# B&R Automation Studio project CombinedLinenSoiledA9KAN (part 17)

#### KanLinkCyclic.st - Cyclic code
```iecst
(********************************************************************
 * COPYRIGHT -- Herbert Kannegiesser GmbH
 ********************************************************************
 * Program: KanLink
 * File: KanLinkCyclic.st
 * Author: stahlhut
 * Created: December 23, 2011
 ********************************************************************
 * Implementation of program WetLink
 ********************************************************************)

(*
	todo
			logger !

	Mögliche Fehler
	1= Configuration kann nicht gelesen werden
	2= Port kann nicht geöffnet werden
	4= Fehler bei UDPSend
	5= Fehler bei UDPRec
*)

PROGRAM _CYCLIC

	// ===========================
	// Logging
	// ===========================

	IF _xRBReady THEN

		CASE _wLogStep OF

			0:
				_ReadRB(wPtrRead := _wPtrRBread, wPtrStart := _wPtrRBstart, wPtrWrite := _wPtrRBwrite);

				IF _ReadRB.wStatus = ERR_OK THEN

					CASE _LogEntry.wErrorNo OF

						0:
							_kgArLogWrite.text := 'OK';

						HLKANLINK_MSG_NO_STRUCDEF:

							_kgArLogWrite.text := 'Create Strucdefinition failed : {##AttrVar1} / {##AttrVar2}';
							_kgArLogWrite.var1 := _LogEntry.lAttr1;

						ELSE

							_kgArLogWrite.text := UINT_TO_STRING(_LogEntry.wErrorNo);
							_kgArLogWrite.text := CONCAT(_kgArLogWrite.text, ' : {##AttrVar1} / {##AttrVar2}');
							_kgArLogWrite.var1 := _LogEntry.lAttr1;
							_kgArLogWrite.var2 := _LogEntry.lAttr2;

					END_CASE

					_wLogStep := 1;

				END_IF

			1:
				_kgArLogWrite();

				IF _kgArLogWrite.status <> ERR_FUB_BUSY THEN

					_wLogStep := 0;

				END_IF

		END_CASE

	END_IF

	IF _wDebIdx >= 0 AND _wDebIdx <= _HLKANLINK_MAX_IDX_DEFSTRUC THEN

		IF _lPtrStrucDef[_wDebIdx] > 0 THEN

			_sDebString ACCESS _lPtrStrucDef[_wDebIdx] + _wDebOffset;

		END_IF

	END_IF

	// =======================================================================
	// =======================================================================

	IF _xInitOK THEN

		IF _xSaveConfig THEN
			KL_SaveConfDO_0(adrName :=ADR('KL_Conf') , adrDaten := ADR(IFhlKanLink.Parameter), len := SIZEOF( IFhlKanLink.Parameter));
			IF KL_SaveConfDO_0.status <> ERR_FUB_BUSY THEN // fertig
				_xSaveConfig := FALSE;
			END_IF;
		END_IF;

		IF EDGEPOS(IFhlKanLink.in.xRun ) THEN
			IF Kanlink.Step = 0 THEN
				Kanlink.Step := 1;
			END_IF;
		END_IF;
		IF EDGENEG(IFhlKanLink.in.xRun) THEN // stoppen
			IF Kanlink.Step <> 0 THEN
				Kanlink.Step := 20;
			END_IF;
		END_IF;

		IF IFhlKanLink.in.xRestart THEN
			Kanlink.Step := 1;
			IFhlKanLink.in.xRestart := 0;
		END_IF;

		IFhlKanLink.xError := (Kanlink.Step = 200);

		CASE Kanlink.Step OF

			0: //nix tun

			100: // Error nr in Logger eintragen

				Kanlink.Step := 200;

			200: // Auf User warten

			1: // init

				Kanlink.KLLib_Init_0(enable := 1, adrServer := ADR(Kanlink),adrInterface := ADR(IFhlKanLink));
				IF Kanlink.KLLib_Init_0.status = ERR_OK THEN
					Kanlink.Step := 10;
				ELSIF Kanlink.KLLib_Init_0.status <> ERR_FUB_BUSY THEN // fehler
					WL_ErrorNr := 10;
					Kanlink.Step := 100;

					IF _xRBReady THEN

						_LogEntryIn.wErrorNo := 10;
						_InsertRB(wPtrStart := _wPtrRBstart, wPtrRead := _wPtrRBread, wPtrWrite := _wPtrRBwrite);

					END_IF

				END_IF;

			10: // Kanlink Run

			20: // Kanlink schliessen
				Kanlink.UdpClose_0(enable := 1);
				Kanlink.UdpClose_0.enable := 1;
				Kanlink.UdpClose_0.ident := Kanlink._uiLastId;
				Kanlink.UdpClose_0;
				IF Kanlink.UdpClose_0.status = 0 THEN
					Kanlink.Step := 0;
				ELSIF Kanlink.UdpClose_0.status = ERR_FUB_BUSY THEN

				ELSE
					Kanlink.Step := 100;
				END_IF;

		END_CASE;

		// hier beenden wenn zyklus nicht erlaubt
		IF  Kanlink.Step <> 10 THEN
			RETURN;
		END_IF;

		//
		// Client Timeout bearbeiten

		Kanlink;

		IF Kanlink.xReturn THEN
			RETURN;
		END_IF;

		IF Kanlink._xGetServerReq THEN  // ServerReq angenommen, bearbeiten

			// antwort zusammenbauen

			// Commandos unter 1000 sind für alle gleich:
			IF Kanlink.ServerData.HeaderV1Rec.Command < 1000 THEN

				CASE Kanlink.ServerData.HeaderV1Rec.Command OF
					0:   // MaschinenInfo Senden: Darf jeder lesen

						Kanlink.ServerData.HeaderV1Send.Command := 1;
						Kanlink.ServerData.HeaderV1Send.dataFormat := 5;
						Kanlink.ServerData.HeaderV1Send.Length := 148;
						Kanlink.ServerData.HeaderV1Send.Tag := Kanlink.ServerData.HeaderV1Rec.Tag;
						Kanlink.ServerData.HeaderV1Send.ReqID := Kanlink.ServerData.HeaderV1Rec.ReqID;

						KLLib_SendData(ADR(Kanlink),ADR(Kanlink.ServerData.MetaInfoResp),SIZEOF(Kanlink.ServerData.MetaInfoResp),ADR(Kanlink.client_address));

					2:   // Response Ping: Darf jeder lesen

						Kanlink.ServerData.HeaderV1Send.Command := 3;
						Kanlink.ServerData.HeaderV1Send.dataFormat := 5;
						Kanlink.ServerData.HeaderV1Send.Length := 17;
						Kanlink.ServerData.HeaderV1Send.Tag := Kanlink.ServerData.HeaderV1Rec.Tag;
						Kanlink.ServerData.HeaderV1Send.ReqID := Kanlink.ServerData.HeaderV1Rec.ReqID;

						KLLib_SendData(ADR(Kanlink),ADR(Kanlink.ServerData.PingResp),SIZEOF(Kanlink.ServerData.PingResp),ADR(Kanlink.client_address));

				END_CASE;

			ELSE
					// >= 1000 sind spezifische Daten

					// Anfrage Konfiguriert?
					// Zur Anfrage Verbindung raussuchen..
					_xIdxFound := FALSE;
					_iIdxFound := 32000;

					//Kanlink.udRecKey	:= SHL(UINT_TO_UDINT( Kanlink.ServerData.HeaderV1Rec.Command),16)  + SHL(USINT_TO_UINT( Kanlink.ServerData.recArea),8) + Kanlink.ServerData.recAddr;

					Kanlink.udRecKey := KL_BuildKey(Command := Kanlink.ServerData.HeaderV1Rec.Command,CmdNr := UINT_TO_USINT( Kanlink.ServerData.HeaderV1Rec.CmdNr AND 16#000F) ,Area := Kanlink.ServerData.recArea,IPAdr:= Kanlink.ServerData.recAddr);
					FOR _i := 0 TO HLKANLINK_MAX_SERVERCONNS  DO

						_ptrIndex ACCESS ADR(Kanlink.ServerListe[_i]);
						_dSrvIf ACCESS _ptrIndex.adrInterface;
						_udRecKey := Kanlink.udRecKey;
						IF _ptrIndex.Adr = 0 THEN // wenn alle das Commando lesen dürfen/ Adresse und Area ausblenden
							_udRecKey := Kanlink.udRecKey AND 16#FFFF_0000;
						END_IF;
						IF _udRecKey = _ptrIndex.Key THEN // Index gefunden, beantworten:
							_xIdxFound := TRUE;
							_iIdxFound := _i;
							EXIT;
						END_IF;
					END_FOR

					_xAdrErr := (_ptrIndex.AdrDataReq = 0) OR (_ptrIndex.AdrDataResp = 0);

					IF ( _xIdxFound = FALSE) OR _xAdrErr THEN // Falls keine gültige Verbindung dann Fehlerframe senden
						// Fehlerframe senden:
						Kanlink.ServerData.HeaderV1Send.Command := Kanlink.ServerData.HeaderV1Rec.Command +1;
						Kanlink.ServerData.HeaderV1Send.dataFormat := 255;
						Kanlink.ServerData.HeaderV1Send.Length := 68;
						Kanlink.ServerData.HeaderV1Send.Tag := Kanlink.ServerData.HeaderV1Rec.Tag;
						Kanlink.ServerData.HeaderV1Send.ReqID := Kanlink.ServerData.HeaderV1Rec.ReqID;

						// Error Frame:
						Kanlink.ServerData.ErrorFrame.ErrorNumber := 2;
						strcpy(ADR(Kanlink.ServerData.ErrorFrame.ErrorText),ADR('request not supported'));

					//	KLLib_SendData(ADR(Kanlink),ADR(Kanlink.ServerData.ErrorFrame),SIZEOF(Kanlink.ServerData.ErrorFrame),ADR(Kanlink.client_address));

				ELSE
						// Empfangene Daten speichern:

						IF NOT( (_dSrvIf.iState <> 0 )   AND _ptrIndex.xReqManually) THEN  // falls Req bereits bearbeitet wird verwerfen
							_ptrIndex.iReqCnt := _ptrIndex.iReqCnt + 1;
							_dSrvIf.iState := 1;
							strcpy(ADR(_ptrIndex.sClientIPAdr),ADR(Kanlink.client_address));
							// todo längenüberprüfung _ptrIndex.ReqLength
							memcpy(_ptrIndex.AdrDataReq,ADR(Kanlink.ServerData.receive_data)+PreHeaderSize+HeaderSize,_ptrIndex.ReqLength);

							_ptrIndex.iReqID := Kanlink.ServerData.HeaderV1Rec.ReqID;
							IF (_ptrIndex.CmdOpt AND KL_optOnReqCall) <> 0 THEN
								KL_OnRecReq(adrReqData := _ptrIndex.AdrDataReq, adrRespData := _ptrIndex.AdrDataResp, adrKanlink := ADR(Kanlink),_ptrIndex.Cmd, adrUserData := IFhlKanLink.Parameter.adrUserTyp );
							END_IF;
							IF _ptrIndex.xReqManually = 0 THEN

								Kanlink.ServerData.HeaderV1Send.Command := _ptrIndex.Cmd + 1;
								Kanlink.ServerData.HeaderV1Send.dataFormat := 5;
								Kanlink.ServerData.HeaderV1Send.Length := UDINT_TO_UINT( _ptrIndex.RespLength);
								Kanlink.ServerData.HeaderV1Send.ReqID := _ptrIndex.iReqID;
								Kanlink.ServerData.HeaderV1Send.CmdNr := _ptrIndex.CmdOpt AND 16#000F;
								_ptrIndex.iConnectionTimer := 0;
								KLLib_SendData(ADR(Kanlink),_ptrIndex.AdrDataResp,_ptrIndex.RespLength,ADR(_ptrIndex.sClientIPAdr));
							END_IF;
						END_IF;

					END_IF;

			END_IF;

			Kanlink._xGetServerReq := FALSE;
			Kanlink.UdpRecv_0.enable := 1;

			RETURN;  // Daten sind versendet. Also Ende.

		END_IF;

		IF Kanlink._xGetClientResp THEN // Response auf ClientReq angekommen

			Kanlink.udRecKey := KL_BuildKey(Command := Kanlink.ServerData.HeaderV1Rec.Command,CmdNr := UINT_TO_USINT( Kanlink.ServerData.HeaderV1Rec.CmdNr AND 16#000F) ,Area := Kanlink.ServerData.recArea,Kanlink.ServerData.recAddr);

			_xIdxFound := FALSE;
			FOR _i := 0 TO HLKANLINK_MAX_CLIENTCONNS DO
				_dClient ACCESS ADR(Kanlink.ClientListe[_i]);
					//Kanlink.udRecKey 	:= SHL(UINT_TO_UDINT( Kanlink.ServerData.HeaderV1Rec.Command),16)  + SHL(USINT_TO_UINT( Kanlink.ServerData.recArea),8) + Kanlink.ServerData.recAddr;

					IF Kanlink.udRecKey = _dClient.Key THEN // Index gefunden, beantworten:
						_xIdxFound := TRUE;
					EXIT;
				END_IF;
			END_FOR

			_xAdrOK := _dClient.AdrDataResp <> 0 ;

			IF _xIdxFound AND _xAdrOK THEN
				_dClient.xReqPending := FALSE;
				IF _dClient.iTimeOutCnt > 0 THEN
					_dClient.iTimeOutCnt := _dClient.iTimeOutCnt - 1;
				END_IF;
				IF _dClient.adrInterface <> 0 THEN
					_dCltIf ACCESS _dClient.adrInterface;
					_dCltIf.iState := 3;
				END_IF;

				memcpy(_dClient.AdrDataResp,ADR(Kanlink.ServerData.receive_data) + PreHeaderSize+HeaderSize,_dClient.RespLength);

		  	END_IF;

			_iCltRespCnt := _iCltRespCnt + 1;
			Kanlink._xGetClientResp := FALSE;

			Kanlink._xSendClient := TRUE; // Daten einsortiert, nix weiter zutun also Clients bearbeiten
			Kanlink.UdpRecv_0.enable := 1;

		END_IF;

		// Überprüfen ob per Hand bearbeitete Requests versendet werden müssen..

		IF  Kanlink.UdpSend_0.enable = 0 THEN
			_xServerFound := 0;

			FOR _i:=0 TO HLKANLINK_MAX_SERVERCONNS  DO
				_ptrIndex ACCESS ADR(Kanlink.ServerListe[_iLastServerIdx]);
				_dSrvIf ACCESS _ptrIndex.adrInterface;
				IF (_ptrIndex.xReqManually AND (_dSrvIf.iState = 2)) THEN
					_xServerFound := 1;

					_iLastServerIdx := _iLastServerIdx + 1; // testen
					IF _iLastCltIdx > HLKANLINK_MAX_SERVERCONNS THEN
						_iLastServerIdx := 0;
					END_IF;
					EXIT;
					END_IF;
					_iLastServerIdx := _iLastServerIdx + 1; // testen
					IF _iLastServerIdx > HLKANLINK_MAX_SERVERCONNS THEN
					_iLastServerIdx := 0;
				END_IF;

			END_FOR;

			IF _xServerFound THEN

				Kanlink.ServerData.HeaderV1Send.Command := _ptrIndex.Cmd + 1;
				Kanlink.ServerData.HeaderV1Send.dataFormat := 5;
				Kanlink.ServerData.HeaderV1Send.Length := UDINT_TO_UINT( _ptrIndex.RespLength);
				Kanlink.ServerData.HeaderV1Send.ReqID := _ptrIndex.iReqID;
				Kanlink.ServerData.HeaderV1Send.CmdNr := _ptrIndex.CmdOpt AND 16#000F;
				_ptrIndex.iConnectionTimer := 0;
				KLLib_SendData(ADR(Kanlink),_ptrIndex.AdrDataResp,_ptrIndex.RespLength,ADR(_ptrIndex.sClientIPAdr));
				_dSrvIf.iState := 0;
				RETURN;
			END_IF;
		END_IF;

		IF Kanlink._xSendClient THEN  // hier den Clienten bearbeiten

			_xCltFound := FALSE;

			FOR _i:=0 TO HLKANLINK_MAX_CLIENTCONNS  DO
				_dClient ACCESS ADR(Kanlink.ClientListe[_iLastCltIdx]);
				IF _dClient.adrInterface <> 0 THEN
					_dCltIf ACCESS _dClient.adrInterface;
				ELSE
					_dCltIf ACCESS ADR(_ifDummy);
				END_IF;
					// gefunden wenn kein ReqPend, Commando <> 0 todo gültige Adresse etc...
				IF _dClient.iCycleTime = 0 THEN
					_xSendNow := (_dCltIf.iState = 1) OR (_dCltIf.iState = 4) ; // falls angetickt oder timeout
				ELSE
					_xSendNow := (_dClient.iCycleWait > _dClient.iCycleTime);
				END_IF;
				IF 	(NOT _dClient.xReqPending) AND (_dClient.Cmd <> 0) AND  _dClient.xActiv AND (_xSendNow)   THEN
		  			_xCltFound := TRUE;
					_iLastCltIdx := _iLastCltIdx + 1; // testen
					IF _iLastCltIdx > HLKANLINK_MAX_CLIENTCONNS THEN
			  			_iLastCltIdx := 0;
					END_IF;
					EXIT;
				END_IF;

				_iLastCltIdx := _iLastCltIdx + 1; // testen
				IF _iLastCltIdx > HLKANLINK_MAX_CLIENTCONNS THEN
		  			_iLastCltIdx := 0;
				END_IF;

			END_FOR;

			IF NOT _xCltFound THEN
				Kanlink._xSendClient := FALSE;
				RETURN;

			ELSE

				// Client gefunden
				_dClient.iCnt := _dClient.iCnt + 1 ;
				_dClient.iReqId := _dClient.iReqId +1;
				_dClient.TimeOutLeft := _dClient.TimeOut;

				IF _dCltIf.iState = 1 THEN // falls über state dann "schnellwiederholung" aktivieren
					_dClient.iTimeOutCnt := 0; // scharf machen für den nächsten versuch
				END_IF;
				_dCltIf.iState := 2;

				Kanlink.ServerData.HeaderV1Send.Command := _dClient.Cmd;
				Kanlink.ServerData.HeaderV1Send.CmdNr := _dClient.CmdOpt AND 16#000F;

				Kanlink.ServerData.HeaderV1Send.dataFormat := 5;
				Kanlink.ServerData.HeaderV1Send.Length := UDINT_TO_UINT( _dClient.ReqLength);
				Kanlink.ServerData.HeaderV1Send.ReqID := _dClient.iReqId;

				KLLib_SendData(ADR(Kanlink),_dClient.AdrDataReq,_dClient.ReqLength,ADR(_dClient.sClientAdr));

				_dClient.xReqPending := TRUE;
				_dClient.iCycleWait := 0;

				Kanlink._xSendClient := FALSE;

				RETURN;

			END_IF;

		END_IF;	// sendClient

	ELSIF IFmnParam.Out.xParamOK AND IFmnEth.Out.xDataValid THEN

		Kanlink.ServerData.MetaInfoResp.KanLink_Hostname := IFmnEth.Out.IP.sHostname;
		Kanlink.ServerData.MetaInfoResp.Machine_type := WSTRING_TO_STRING(IFmnParam.Out.HeaderVersion.utfMachineType);
		Kanlink.ServerData.MetaInfoResp.DataModelTimeStamp := IFmnParam.Out.HeaderVersion.dtTimestamp;
		Kanlink.ServerData.MetaInfoResp.DataModelVersion := IFmnParam.Out.HeaderVersion.wVersion;

		Kanlink.ServerData.PingResp.KanLink_Hostname := IFmnEth.Out.IP.sHostname;

		_xInitOK := TRUE;

	END_IF

END_PROGRAM
```

#### KanLinkInit.st - Initialization code
```iecst
(********************************************************************
 * COPYRIGHT -- Herbert Kannegiesser GmbH
 ********************************************************************
 * Program: KanLink
 * File: KanLinkInit.st
 * Author: stahlhut
 * Created: December 23, 2011
 ********************************************************************
 * Implementation of program KanLink
 ********************************************************************)

PROGRAM _INIT

	// Packet-Version auslesen mit MO_ver aus SYS_lib und für den Additional Status zur Verfügung stellen

	_sPkgName := 'hlKanLink';

	IF ( MO_ver(ADR(_sPkgName), 0, ADR(_VerStruc)) = 0 ) THEN

		brsmemcpy(ADR(hlKanLinkStatAd.sPkgVersion), ADR(_VerStruc.version), SIZEOF(_VerStruc.version));

	ELSE

		hlKanLinkStatAd.sPkgVersion := '---';

	END_IF

	_xInitOK := FALSE;

	// nötige adressen initialisieren:
	Kanlink.adrSelf := ADR(Kanlink);
	Kanlink.CfgServer.adrKanlink := ADR(Kanlink);
	Kanlink.CfgClient.adrKanlink := ADR(Kanlink);

	FOR _i := 0 TO HLKANLINK_MAX_SERVERCONNS DO
		Kanlink.ServerListe[_i].adrInterface := ADR(IFhlKanLink.Server[_i]);
		KLLib_ReadServerPara(ADR(Kanlink.ServerListe[_i]), ADR( IFhlKanLink.Parameter.Server[_i]));
	END_FOR;

	FOR _i := 0 TO HLKANLINK_MAX_CLIENTCONNS DO
		KLLib_ReadClientPara(ADR(Kanlink.ClientListe[_i]),ADR(IFhlKanLink.Parameter.Client[_i]),ADR(Kanlink));
		Kanlink.ClientListe[_i].TimeOut := 140;
		Kanlink.ClientListe[_i].adrInterface := ADR(IFhlKanLink.Parameter.Client[_i]);
	END_FOR;

	// Create Log
	//****************************************************************************************************************
	// Log erzeugen
	//****************************************************************************************************************

	_kgArLogWrite.enable := TRUE;
	_kgArLogWrite.ident := 0;
	_kgArLogWrite.errornr := 50010;

	_AsArLogCreate(enable := TRUE, pName := ADR('hlKanLinkL'), len := 4096*1, memType := arlogUSRROM);

	IF _AsArLogCreate.status = ERR_OK THEN

		_kgArLogWrite.ident := _AsArLogCreate.ident;

	ELSIF _AsArLogCreate.status = arlogERR_EXISTING THEN

		_AsArLogGetInfo(enable := TRUE, pName := ADR('hlKanLinkL'));

		IF _AsArLogGetInfo.status = ERR_OK THEN

			_kgArLogWrite.ident := _AsArLogGetInfo.ident;

		END_IF

	END_IF

	//****************************************************************************************************************
	// Ringbuffer for Logs
	//****************************************************************************************************************

	_kgRBcreateKanLinklog(sName := '_klLogrb', bMemType := doUSRRAM, wCntEntry := 10, lLenEntry := SIZEOF(_LogEntry), wPtrWrite := _wPtrRBwrite, wPtrRead := _wPtrRBread, wPtrStart := _wPtrRBstart);

	IF _kgRBcreateKanLinklog.wStatus = ERR_OK THEN

		_wPtrRBloc := 0;

		_xRBReady := TRUE;

		_InsertRB.doIdent := _kgRBcreateKanLinklog.doIdent;
		_InsertRB.doLen := _kgRBcreateKanLinklog.doLen;
		_InsertRB.lLenEntry := SIZEOF(_LogEntry);
		_InsertRB.pEntry := ADR(_LogEntryIn);

		_ReadRB.doIdent := _kgRBcreateKanLinklog.doIdent;
		_ReadRB.doLen := _kgRBcreateKanLinklog.doLen;
		_ReadRB.lLenEntry := SIZEOF(_LogEntry);
		_ReadRB.pEntry := ADR(_LogEntry);

	ELSE

		_kgArLogWrite.logLevel := arlogLEVEL_INFO;
		_kgArLogWrite.text := 'Create Ringbuffer: {##AttrVar1}';
		_kgArLogWrite.var1 := _kgRBcreateKanLinklog.wStatus;
		_kgArLogWrite.var2 := 0;
		_kgArLogWrite();

	END_IF

	_wLogStep := 0;

	// Create StructureDescriptions
	//****************************************************************************************************************
	// Speicher allokoieren
	//****************************************************************************************************************

	_MemPartCreate(enable := TRUE, len := 8000);

	_LogEntryIn.wErrorNo := HLKANLINK_MSG_NO_STRUCDEF;

	IF _MemPartCreate.status = ERR_OK THEN

		_lTempMemIdent := _MemPartCreate.ident;

		_MemPartCreate(enable := TRUE, len := 8000);

		IF _MemPartCreate.status = ERR_OK THEN

			_lMemIdent := _MemPartCreate.ident;

			_MemAllocTemp(enable := TRUE, ident := _lTempMemIdent, len := 7500);

			IF _MemAllocTemp.status = ERR_OK THEN

				_lAdr := _MemAllocTemp.mem;
				_lLen := _MemAllocTemp.len;

				_wStatus := KLLib_CreateStrucDef(lPtrAdr := ADR(_lAdr), lPtrLen := ADR(_lLen), sRootName := 'hlKanLink:Kanlink.ServerData.MetaInfoResp', sItemName := '', lDataAdr := 0);

				IF _wStatus = ERR_OK THEN

					_MemAlloc(enable := TRUE, ident := _lMemIdent, len := _MemAllocTemp.len - _lLen);

					IF _MemAlloc.status = ERR_OK THEN

						_lPtrStrucDef[_HLKANLINK_IDX_STRUCDEF_RESP_0] := _MemAlloc.mem;
						_lPtrStrucLen[_HLKANLINK_IDX_STRUCDEF_RESP_0] := _MemAlloc.len;

						brsmemcpy(_MemAlloc.mem, _MemAllocTemp.mem, _MemAlloc.len);

						_MemFreeTemp(enable := TRUE, ident := _lTempMemIdent, mem := _MemAllocTemp.mem );

					ELSE

						_LogEntryIn.lAttr1 := _MemAlloc.status;
						_InsertRB(wPtrStart := _wPtrRBstart, wPtrRead := _wPtrRBread, wPtrWrite := _wPtrRBwrite);

					END_IF

				ELSE

					_LogEntryIn.lAttr1 := _wStatus;
					_InsertRB(wPtrStart := _wPtrRBstart, wPtrRead := _wPtrRBread, wPtrWrite := _wPtrRBwrite);

				END_IF

			ELSE

				_LogEntryIn.lAttr1 := _MemAllocTemp.status;
				_InsertRB(wPtrStart := _wPtrRBstart, wPtrRead := _wPtrRBread, wPtrWrite := _wPtrRBwrite);

			END_IF

		ELSE

			_LogEntryIn.lAttr1 := _MemPartCreate.status;
			_InsertRB(wPtrStart := _wPtrRBstart, wPtrRead := _wPtrRBread, wPtrWrite := _wPtrRBwrite);

		END_IF

	ELSE

		_LogEntryIn.lAttr1 := _MemPartCreate.status;
		_InsertRB(wPtrStart := _wPtrRBstart, wPtrRead := _wPtrRBread, wPtrWrite := _wPtrRBwrite);

	END_IF

END_PROGRAM
```

#### KanLink.typ - Local data types
```iecst
(********************************************************************
 * COPYRIGHT -- Herbert Kannegiesser GmbH
 ********************************************************************
 * Program: WetLink
 * File: WetLink.typ
 * Author: stahlhut
 * Created: December 23, 2011
 ********************************************************************
 * Local data types of program WetLink
 ********************************************************************)

TYPE
	Server_typ : 	STRUCT  (*UDP Server Variables*)
		sStep : UINT; (*UDP Server Step Variable*)
		client_address : STRING[20]; (*Address of the client connection to the Server*)
		UdpOpen_0 : UdpOpen; (*AsUDP.UdpOpen FUB*)
		UdpSend_0 : UdpSend; (*AsUDP.UdpSend FUB*)
		UdpRecv_0 : UdpRecv; (*AsUDP.UdpRecv FUB*)
		UdpClose_0 : UdpClose; (*AsUDP.UdpClose FUB*)
		iPort : UINT;
		sIF : STRING[10];
	END_STRUCT;
	ErrLog_typ : 	STRUCT
		wErrorNo : UINT;
		lAttr1 : UDINT;
		lAttr2 : UDINT;
	END_STRUCT;
END_TYPE
```

#### KanLink.var - Local variables
```iecst
(********************************************************************
 * COPYRIGHT -- Herbert Kannegiesser GmbH
 ********************************************************************
 * Program: WetLink
 * File: WetLink.var
 * Author: stahlhut
 * Created: December 23, 2011
 ********************************************************************
 * Local variables of program WetLink
 ********************************************************************)
VAR
	_xIdxFound : BOOL;
	_ptrIndex : REFERENCE TO KL_ServerListe_typ;
	_i : UINT;
	_iCltRespCnt : INT;
	_xCltFound : BOOL;
	_xInitOK : BOOL;
	_kgArLogWrite : kgArLogWrite;
	_AsArLogCreate : AsArLogCreate;
	_AsArLogGetInfo : AsArLogGetInfo;
	_sLogEntry : STRING[63];
	_wPtrRBwrite : UINT;
	_wPtrRBread : UINT;
	_wPtrRBstart : UINT;
	_kgRBcreateKanLinklog : kgRBcreate;
	_wPtrRBloc : UINT;
	_xRBReady : BOOL;
	_InsertRB : kgRBinsert;
	_ReadRB : kgRBread;
	_sLogEntryIn : STRING[63];
	_LogEntry : ErrLog_typ;
	_LogEntryIn : ErrLog_typ;
	_wLogStep : UINT;
	_MemPartCreate : AsMemPartCreate;
	_lTempMemIdent : UDINT;
	_lMemIdent : UDINT;
	_MemAlloc : AsMemPartAllocClear;
END_VAR
VAR RETAIN
	_iLastCltIdx : UINT;
END_VAR
VAR
	_dClient : REFERENCE TO KL_ClientListe_typ;
	_xAdrErr : BOOL;
	_iIdxFound : INT;
	_xAdrOK : BOOL;
	WL_ErrorNr : UINT;
	KL_SaveConfDO_0 : KL_SaveConfDO;
	_xSaveConfig : BOOL;
	_iLastServerIdx : UINT;
	_xServerFound : BOOL;
	_dSrvIf : REFERENCE TO IF_Server;
	_udRecKey : UDINT;
	_dCltIf : REFERENCE TO IF_Client_typ;
	_ifDummy : IF_Client_typ;
	_xSendNow : BOOL;
	Kanlink : KanLink_FB;
	_sPkgName : STRING[11];
	_VerStruc : MoVerStruc_typ;
	_lAdr : UDINT;
	_lLen : UDINT;
	_wStatus : UINT;
	_MemAllocTemp : AsMemPartAllocClear;
END_VAR
VAR CONSTANT
	_HLKANLINK_IDX_STRUCDEF_RESP_0 : UINT := 1;
END_VAR
VAR
	_lPtrStrucDef : ARRAY[0..5] OF UDINT;
	_lPtrStrucLen : ARRAY[0..5] OF UDINT;
	_MemFreeTemp : AsMemPartFree;
	_wDebIdx : UINT;
END_VAR
VAR CONSTANT
	_HLKANLINK_MAX_IDX_DEFSTRUC : UINT := 5;
END_VAR
VAR
	_sDebString : REFERENCE TO STRING[31];
	_wDebOffset : UINT;
END_VAR
```

### Library Logical/Mewa/KGFramework/Pkg_hlKanLink/KanLinkLib (IEC) - KanlinkHilfsfunktionen
Depends on: AsUDP, asstring, AsARCfg, brsystem, sys_lib, AsArLog, AsIODiag, AsETH, DataObj, KL_UserLib, KGstdLib

#### KanLinkLib.typ - Exported data types
```iecst
(********************************************************************
 * COPYRIGHT -- Herbert Kannegiesser GmbH
 ********************************************************************
 * Library: WetLinkLib
 * File: WetLinkLib.typ
 * Author: stahlhut
 * Created: January 06, 2012
 ********************************************************************
 * Data types of library WetLinkLib
 ********************************************************************)
(*Interne Strukturen*)

TYPE
	udint_array_typ : 	STRUCT
		a : USINT;
		b : USINT;
		c : USINT;
		d : USINT;
	END_STRUCT;
	ServerDataTyp : 	STRUCT  (*Datatyp for global Variables*)
		receive_data : ARRAY[0..8191]OF USINT; (*Data which has been received*)
		send_data : ARRAY[0..8191]OF USINT; (*Data which should be sent*)
		PreHeaderSend : PreHeader_Typ;
		PreHeaderRec : PreHeader_Typ;
		HeaderV1Send : HeaderV1_Typ;
		HeaderV1Rec : HeaderV1_Typ;
		MetaInfoResp : KLresp0_MetaInfo_typ;
		ErrorFrame : KL_Error_Frame_typ;
		PingReq : KLreq2_Ping_typ;
		PingResp : KLresp2_Ping_typ;
		recArea : USINT; (*Bereich des Client*)
		recAddr : USINT; (*Adresse des Client*)
	END_STRUCT;
	PreHeader_Typ : 	STRUCT
		Magic : UDINT; (*MagicNr*)
		HeaderVersion : UINT; (*Headerversion*)
		Tag : UINT; (*Reserve*)
	END_STRUCT;
	HeaderV1_Typ : 	STRUCT
		ReqID : UINT;
		dataFormat : UINT;
		Command : UINT;
		Length : UINT;
		CmdNr : UINT;
		CmdTag : UINT; (*Unterschiedliche Parameter zum Command*)
		Tag : UDINT; (*Reserve/Spezial*)
	END_STRUCT;
END_TYPE

(*Kommandos*)

TYPE
	PartBatchData_typ : 	STRUCT
		sCustomNo : STRING[11];
		wCustomWeight : UINT;
	END_STRUCT;
	BatchData_typ : 	STRUCT
		dtTimeStamp : DATE_AND_TIME;
		bTypeBatchNo : USINT;
		bCntCustomers : USINT;
		wTotalWeight : UINT;
		bBatchNo : ARRAY[0..15]OF USINT;
		sCategory : STRING[11];
		utfMark : ARRAY[0..31]OF UINT;
		bCustom : ARRAY[0..11]OF USINT;
		PartBatch : ARRAY[0..7]OF PartBatchData_typ;
	END_STRUCT;
	KL_Error_Frame_typ : 	STRUCT
		Version : UINT;
		ErrorNumber : UINT;
		ErrorText : STRING[63];
	END_STRUCT;
	KLresp0_MetaInfo_typ : 	STRUCT
		KanLink_Hostname : STRING[15];
		Machine_type : STRING[15];
		SoftwareNo : STRING[15];
		SoftwareVersion : STRING[15];
		DataModelTimeStamp : DATE_AND_TIME;
		DataModelVersion : UINT;
		TimeZone : UINT;
		SommerTime : UINT;
	END_STRUCT;
	KLreq2_Ping_typ : 	STRUCT
		KanLink_Hostname : STRING[15];
	END_STRUCT;
	KLresp2_Ping_typ : 	STRUCT
		KanLink_Hostname : STRING[15];
		FrameVersion : USINT;
	END_STRUCT;
	KL_BTxf_typ : 	STRUCT  (*Batch Transfer Server*)
		Req : KLreq1000_BTH_typ;
		Resp : KLresp1000_BTH_typ;
	END_STRUCT;
	KL_BI_typ : 	STRUCT
		Req : KLreq1002_Info_typ;
		Resp : KLresp1002_Info_typ;
	END_STRUCT;
	KL_ServerListe_typ : 	STRUCT
		Cmd : UINT;
		CmdOpt : UINT;
		Adr : UINT;
		Area : UINT;
		pRespStr : UDINT; (*Adresse des Resp String*)
		pReqStr : UDINT; (*Adresse des Req String*)
		AdrDataReq : UDINT;
		ReqLength : UDINT; (*Länge Request Daten*)
		AdrDataResp : UDINT;
		RespLength : UDINT; (*Länge Response Daten*)
		Key : UDINT; (*Suchschlüssel/ Darf nicht doppelt vorkommen== Konfigurierungsfehler*)
		xConnected : BOOL; (*Falls Commando 2s nicht angefragt wird ist verbindung unterbrochen*)
		iConnectionTimer : UINT; (*Der Zugehörige Zähler / Timer*)
		adrParameter : UDINT; (*Adresse der Parameter*)
		sClientIPAdr : STRING[20];
		iReqCnt : UINT;
		xReqManually : BOOL;
		iReqID : UINT;
		iCfgStatus : UINT;
		adrInterface : UDINT;
		xActiv : BOOL;
	END_STRUCT;
	KL_ClientListe_typ : 	STRUCT
		RecCmd : UINT; (*Rec Command nr*)
		Cmd : UINT; (*Send Command nr*)
		CmdOpt : UINT; (*SendeOptionen Senden Nr des Commando etc*)
		Adr : UINT;
		Area : UINT;
		Key : UDINT;
		pResp : UDINT; (*Adresse des Namen der Response Struktur*)
		pReq : UDINT; (*Adresse des Namen der Request Struktur*)
		AdrDataReq : UDINT;
		AdrDataResp : UDINT;
		ReqLength : UDINT;
		RespLength : UDINT;
		TimeOut : UINT;
		TimeOutLeft : UINT;
		xError : BOOL;
		iCycleWait : UINT;
		iCycleTime : UINT;
		xDataRec : BOOL;
		iReqId : UINT;
		sClientAdr : STRING[20];
		xReqPending : BOOL;
		iTimeOutCnt : UINT;
		xActiv : BOOL;
		iCnt : UINT;
		xConnected : BOOL; (*True wenn Verbindung aktiv und läuft*)
		iTimeOutCnt_Summe : UINT;
		adrInterface : UDINT;
		adrParameter : UDINT; (*Adresse der Parameter*)
	END_STRUCT;
	KLreq1000_BTH_typ : 	STRUCT
		xHready : BOOL;
		xHreadyForLoad : BOOL;
		xHbatchReceived : BOOL;
		xHtransferzoneOccupied : BOOL;
		xHreqCtrlTransfer : BOOL;
		xHtransferRunning : BOOL;
		xHwaitingForTransfer : BOOL;
		xHshiftBatches : BOOL;
		wHstate : UINT;
		xHcmdAutomatic : BOOL;
		xHreserve : ARRAY[1..5]OF BOOL;
		wTimeToReadyForLoad : UINT;
		wRemainProctime : UINT; (*Remaining Processtime / Verbleibende Prozesszeit*)
	END_STRUCT;
	KLresp1000_BTH_typ : 	STRUCT
		xHsCmdFinishProcess : BOOL;
		xHsReqForUnload : BOOL;
		xHsUnloading : BOOL;
		xHsReqCtrlTransfer : BOOL;
		xHsTransferRunning : BOOL;
		xHsRes : BOOL;
		wState : UINT;
		xCmdAuto : BOOL;
		xCmdStartProcess : BOOL;
		xHsDataValid : BOOL;
		xHsRes2 : ARRAY[0..2]OF BOOL;
		wCntLoads : UINT;
		BatchData : BatchData_typ;
	END_STRUCT;
	KLreq1002_Info_typ : 	STRUCT
		wCntPositions : UINT;
		wNoOfPosition : ARRAY[0..5]OF UINT;
		wRes : UINT;
	END_STRUCT;
	KLresp1002_Info_typ : 	STRUCT
		wCntPositions : UINT;
		wNoOfPositions : ARRAY[0..5]OF UINT;
		wRes : UINT;
		BatchData : ARRAY[0..5]OF BatchData_typ;
	END_STRUCT;
	KLresp30010_SH_typ : 	STRUCT
		MachineNo : STRING[15];
		State : UINT;
		RouteState : ARRAY[1..20]OF UINT;
		WetAccState : ARRAY[1..10]OF UINT;
		WetAccNiveau_mm : ARRAY[1..10]OF UINT;
		WetAccNiveau_rel : ARRAY[1..10]OF UINT;
		WetAccNiveau_Liter : ARRAY[1..10]OF UINT;
		WetAccTemp : ARRAY[1..10]OF UINT;
		WetAccMinLvlOK : ARRAY[1..10]OF UINT;
		WetAccMaxLvlOK : ARRAY[1..10]OF UINT;
	END_STRUCT;
	KLreq30010_SH_typ : 	STRUCT
		MachineNo : STRING[15];
		State : UINT;
		Handshake : BOOL;
		Route : ARRAY[1..20]OF USINT;
		TankTemp : ARRAY[1..10]OF UINT;
	END_STRUCT;
	KL_SiloData_typ : 	STRUCT
		Req : KLreq30010_SH_typ;
		Resp : KLresp30010_SH_typ;
	END_STRUCT;
END_TYPE

(*Interfacing*)

TYPE
	KL_Parameter_typ : 	STRUCT
		Server : ARRAY[0..HLKANLINK_MAX_SERVERCONNS]OF KL_ServerPar_typ;
		Client : ARRAY[0..HLKANLINK_MAX_CLIENTCONNS]OF KL_ClientPar_typ;
		adrUserTyp : UDINT;
	END_STRUCT;
	KL_ClientPar_typ : 	STRUCT
		Name : STRING[15];
		Adr : UINT;
		Cmd : UINT;
		CmdOpt : UINT; (*Bits 0..3 = Nummer des Clients*)
		Area : UINT;
		CycleTime : UINT;
		sReq : STRING[80];
		sResp : STRING[80];
	END_STRUCT;
	KL_ServerPar_typ : 	STRUCT
		Name : STRING[15];
		Adr : UINT;
		Cmd : UINT;
		CmdOpt : UINT; (*Bits 0..3 = Nummer der Verbindung*)
		Area : UINT;
		TimeOut : UINT;
		sReq : STRING[80];
		sResp : STRING[80];
	END_STRUCT;
	IF_ServerOutTyp : 	STRUCT
		xConnected : BOOL;
		iCfgState : UINT; (*0 = ConfOK*)
	END_STRUCT;
	IF_Server : 	STRUCT
		iState : UINT;
		out : IF_ServerOutTyp;
	END_STRUCT;
	IF_ClientOut_typ : 	STRUCT
		xConnected : BOOL;
	END_STRUCT;
	IF_Client_typ : 	STRUCT
		out : IF_ClientOut_typ;
		iState : UINT;
	END_STRUCT;
	IFhlKanLink_Typ : 	STRUCT
		in : IF_KL_Control_in_typ;
		Server : ARRAY[0..HLKANLINK_MAX_SERVERCONNS]OF IF_Server;
		Client : ARRAY[0..HLKANLINK_MAX_CLIENTCONNS]OF IF_Client_typ;
		Parameter : KL_Parameter_typ;
		xError : BOOL; (*Kanlink in Störung*)
	END_STRUCT;
	IF_KL_Control_in_typ : 	STRUCT
		xRun : BOOL; (*Rise= Starten Kanlink /fall = stoppen Kanlink*)
		xRestart : BOOL;
	END_STRUCT;
	IF_KL_Control_out_typ : 	STRUCT
		iError : UINT;
		iServerError : ARRAY[0..HLKANLINK_MAX_SERVERCONNS]OF UINT;
		iClientError : ARRAY[0..HLKANLINK_MAX_CLIENTCONNS]OF UINT;
		iStep : UINT; (*Statemachine KanLink*)
	END_STRUCT;
END_TYPE
```

#### KanLinkLib.var - Exported constants
```iecst
(********************************************************************
 * COPYRIGHT -- Herbert Kannegiesser GmbH
 ********************************************************************
 * Library: WetLinkLib
 * File: WetLinkLib.var
 * Author: stahlhut
 * Created: January 06, 2012
 ********************************************************************
 * Constants of library WetLinkLib
 ********************************************************************)
VAR CONSTANT
	MagicNr : UDINT := 16#B16B00B5;
	PreHeaderSize : UDINT := 8;
	HeaderSize : UDINT := 16;
	KL_optReqManually : UINT := 16#8000;
	KL_optOnReqCall : UINT := 16#4000;
	KLLIB_MSG_NULL_POINTER : UINT := 60000;
	KLLIB_MSG_NOT_ENOUGH_MEM : UINT := 60001;
	KLLIB_MSG_VAR_ERROR : UINT := 60002;
END_VAR
```

#### KanLinkLib.fun - Exported functions and function blocks
```iecst
(********************************************************************
 * COPYRIGHT -- Herbert Kannegiesser GmbH
 ********************************************************************
 * Library: WetLinkLib
 * File: WetLinkLib.fun
 * Author: stahlhut
 * Created: January 06, 2012
 ********************************************************************
 * Functions and function blocks of library WetLinkLib
 ********************************************************************)

FUNCTION_BLOCK KanLink_FB (*TODO: Add your comment here*)
	VAR_INPUT
		UdpClose_0 : UdpClose;
		Step : UINT; (*state machine*)
		client_address : STRING[20]; (*Speichern der Receiver Adresse*)
		UdpOpen_0 : UdpOpen;
		UdpSend_0 : UdpSend;
		UdpRecv_0 : UdpRecv;
		iPort : UINT; (*Port nr (23500)*)
		sIF : STRING[10]; (*Interface Ethernet*)
		ServerData : ServerDataTyp;
		ServerListe : ARRAY[0..HLKANLINK_MAX_SERVERCONNS] OF KL_ServerListe_typ; (*Erlaubte Daten Server*)
		_xOpenPort : BOOL;
		_xSendClient : BOOL;
		_xGetClientResp : BOOL;
		_xGetServerReq : BOOL;
		_uiLastId : UDINT;
		CanReturn : BOOL;
		ClientListe : ARRAY[0..HLKANLINK_MAX_CLIENTCONNS] OF KL_ClientListe_typ;
		adrSelf : UDINT; (*Eigene Adresse, zum weiterleiten an Function/Function Block*)
		_offset : UDINT; (*Offset zum Berechnen der Sendelänge*)
		_SendLen : UDINT; (*Sendelänge*)
		DoCommand : UINT;
		sNetID : STRING[15];
		udNetID : UDINT;
		KLLib_Init_0 : KLLib_Init;
		_iCycleTime : UINT;
		adrInterface : UDINT;
		ErrorNr : UINT;
		udRecKey : UDINT;
		CfgClient : KLLib_CfgClient;
		CfgServer : KLLib_CfgServer;
	END_VAR
	VAR_OUTPUT
		xReturn : BOOL;
	END_VAR
	VAR
		_dPrehead : REFERENCE TO PreHeader_Typ;
		_dHead : REFERENCE TO HeaderV1_Typ;
		_udArr : REFERENCE TO udint_array_typ;
		_dRecAdr : UDINT;
		_xPreheadOK : BOOL;
		_xVersionOK : BOOL;
	END_VAR
END_FUNCTION_BLOCK

FUNCTION KLLib_ClientTimer : BOOL (*Bearbeitet Timeout und Cycletime (Zähler)*)
	VAR_INPUT
		Srv : REFERENCE TO KanLink_FB;
		_iCycleTime : UINT;
	END_VAR
	VAR
		_dClient : REFERENCE TO KL_ClientListe_typ;
		_i : UINT;
		_dServer : REFERENCE TO KL_ServerListe_typ;
		_dInterface : REFERENCE TO IF_Client_typ;
		_dSrvIf : REFERENCE TO IF_Server;
	END_VAR
END_FUNCTION

FUNCTION KLLib_GetPVAdr : UDINT (*Adresse der PV ermitteln (Server)*)
	VAR_INPUT
		ServerItem : REFERENCE TO KL_ServerListe_typ;
	END_VAR
	VAR
		iStat : INT;
	END_VAR
END_FUNCTION

FUNCTION KLLib_SendData : UDINT (*TODO: Add your comment here*)
	VAR_INPUT
		Srv : REFERENCE TO KanLink_FB;
		SendAdr : UDINT;
		SendLen : UDINT;
		pDestination : UDINT; (*Adresse des Zielstrings*)
	END_VAR
END_FUNCTION

FUNCTION KLLib_ReadServerPara : UDINT (*TODO: Add your comment here*)
	VAR_INPUT
		adrServerItem : UDINT;
		adrParaItem : UDINT;
	END_VAR
	VAR
		_xError : BOOL;
		dServer : REFERENCE TO KL_ServerListe_typ;
		dPara : REFERENCE TO KL_ServerPar_typ;
	END_VAR
END_FUNCTION

FUNCTION KLLib_ReadClientPara : UDINT (*TODO: Add your comment here*)
	VAR_INPUT
		adrClientItem : UDINT;
		adrParaItem : UDINT;
		adrServer : UDINT;
	END_VAR
	VAR
		_xError : BOOL;
		dClient : REFERENCE TO KL_ClientListe_typ;
		dPara : REFERENCE TO KL_ClientPar_typ;
		_udArr : REFERENCE TO udint_array_typ;
		_udAdr : UDINT;
		dServer : REFERENCE TO KanLink_FB;
		_udNetId : REFERENCE TO udint_array_typ;
	END_VAR
END_FUNCTION

FUNCTION KLLib_InitCltPV : UDINT (*TODO: Add your comment here*)
	VAR_INPUT
		dclt : REFERENCE TO KL_ClientListe_typ;
	END_VAR
	VAR
		iStat : UINT;
	END_VAR
END_FUNCTION

FUNCTION_BLOCK KLLib_Init (*TODO: Add your comment here*)
	VAR_INPUT
		enable : BOOL;
		adrServer : UDINT;
		adrInterface : UDINT;
	END_VAR
	VAR_OUTPUT
		status : UINT;
	END_VAR
	VAR
		_bStep : INT;
		_dServer : REFERENCE TO KanLink_FB;
		GetEthPort_0 : kgGetEthPort;
		CfgGetIPAddr_0 : CfgGetIPAddr;
		RTInfo_0 : RTInfo;
		_i : INT;
		_dIf : REFERENCE TO IFhlKanLink_Typ;
	END_VAR
END_FUNCTION_BLOCK

FUNCTION KL_BuildKey : UDINT
	VAR_INPUT
		Command : UINT;
		CmdNr : USINT;
		Area : USINT;
		IPAdr : USINT;
	END_VAR
END_FUNCTION

FUNCTION_BLOCK KLLib_CfgClient (*Configuriert einen Kanlink Client*)
	VAR_INPUT
		adrKanlink : UDINT;
		ClientIndex : UINT;
		adrName : UDINT;
		IPAdr : USINT;
		Area : USINT;
		CmdOpt : UINT;
		Cmd : UINT;
		CycleTime : UINT;
		adrSReq : UDINT;
		adrSResp : UDINT;
	END_VAR
	VAR_OUTPUT
		status : UINT;
	END_VAR
	VAR
		_dKL : REFERENCE TO KanLink_FB;
		_dCltPar : REFERENCE TO KL_ClientPar_typ;
		_iret : UDINT;
	END_VAR
END_FUNCTION_BLOCK

FUNCTION_BLOCK KLLib_CfgServer (*Configuriert einen Kanlink Server*)
	VAR_INPUT
		adrKanlink : UDINT;
		ServerIndex : UINT;
		adrName : UDINT;
		IPAdr : USINT;
		Area : USINT;
		CmdOpt : UINT;
		Cmd : UINT;
		TimeOut : UINT;
		adrSReq : UDINT;
		adrSResp : UDINT;
	END_VAR
	VAR_OUTPUT
		status : UINT;
	END_VAR
	VAR
		_dKL : REFERENCE TO KanLink_FB;
		_dSrvPar : REFERENCE TO KL_ServerPar_typ;
		_iret : UDINT;
	END_VAR
END_FUNCTION_BLOCK

FUNCTION KLLib_CreateStrucDef : UINT (*Erzeuge eine Strukturdefinition zu einer Variablen*)
	VAR_INPUT
		lPtrAdr : UDINT;
		lPtrLen : UDINT;
		sRootName : STRING[127];
		sItemName : STRING[31];
	END_VAR
	VAR
		_wStatus : UINT;
		_sPvName : STRING[127];
		_lDataType : UDINT;
		_lDataLen : UDINT;
		_wDataDimension : UINT;
		_sLine : STRING[127];
		_sValueLen : STRING[11];
		_lOffset : UDINT;
		_lAdr : REFERENCE TO UDINT;
		_lLen : REFERENCE TO UDINT;
		_sValueDim : STRING[5];
		_sValueOffs : STRING[11];
		_iStringlen : INT;
		_i : UINT;
		_sItemName : STRING[31];
		_sType : ARRAY[1..23] OF STRING[15] := ['BOOL','SINT','INT','DINT','USINT','UINT','UDINT','REAL','STRING','ULINT','DATE_AND_TIME','TIME','DATE','LREAL','','TIME_OF_DAY','BYTE','WORD','DWORD','LWORD','WSTRING','','LINT'];
	END_VAR
	VAR_INPUT
		lDataAdr : UDINT;
	END_VAR
	VAR
		_lDataAdr : UDINT;
	END_VAR
END_FUNCTION

FUNCTION KLLib_WriteStrucDefLine : UINT (*Übertrage einen String als Zeile in den Speicher*)
	VAR_INPUT
		lPtrLine : UDINT;
		lPtrAdr : UDINT;
		lPtrLen : UDINT;
	END_VAR
	VAR
		_lAdr : REFERENCE TO UDINT;
		_lLen : REFERENCE TO UDINT;
		_iStringlen : INT;
		_sLine : REFERENCE TO STRING[127];
	END_VAR
END_FUNCTION
```

#### KLLib_CfgClient.st - Configuriert einen Kanlink Server
```iecst
(********************************************************************
 * COPYRIGHT -- Herbert Kannegiesser GmbH
 ********************************************************************
 * Library: KanLinkLib
 * File: KLLib_CfgServer.st
 * Author: stahlhut
 * Created: February 01, 2012
 ********************************************************************
 * Implementation of library KanLinkLib
 ********************************************************************)

(* Configuriert einen Kanlink Client *)
FUNCTION_BLOCK KLLib_CfgClient
	// überprüfen
	IF (adrKanlink = 0) OR (adrSReq = 0) OR (adrSResp = 0) OR (adrName = 0)  THEN
		status := 1; // Fehler 1 adressen fehler
		RETURN;
	END_IF;
	IF (ClientIndex > HLKANLINK_MAX_CLIENTCONNS) THEN
		status := 2; // Fehler Index zu gross
		RETURN;
	END_IF;

	_dKL ACCESS adrKanlink;
	IF _dKL.ClientListe[ClientIndex].adrParameter = 0 THEN
		status := 3; // fehler Kanlink / fehlende init der adressen Interface
		RETURN;
	END_IF;

	IF CycleTime < 200 THEN
		CycleTime := 1000;
	END_IF;

	_dCltPar ACCESS _dKL.ClientListe[ClientIndex].adrParameter;
	_dCltPar.Adr := IPAdr;
	_dCltPar.Area := Area;
	_dCltPar.Cmd := Cmd;
	_dCltPar.CmdOpt := CmdOpt;
	memcpy(ADR( _dCltPar.Name ),adrName,15);
	memcpy(ADR(_dCltPar.sReq),adrSReq,80);
	memcpy(ADR(_dCltPar.sResp),adrSResp,80);
	_dCltPar.CycleTime := CycleTime;

	_iret := KLLib_ReadClientPara(ADR(_dKL.ClientListe[ClientIndex]),(_dKL.ClientListe[ClientIndex].adrParameter),adrKanlink);

	IF ( _iret <> 0 ) THEN
		_dKL.ClientListe[ClientIndex].xActiv := 0;
		status := 4;
	ELSE
		_dKL.ClientListe[ClientIndex].xActiv := (_dKL.ClientListe[ClientIndex].Cmd <> 0);
		status := 0; // mit ok beenden
	END_IF;

END_FUNCTION_BLOCK
```

#### KLLib_CfgServer.st - Configuriert einen Kanlink Server
```iecst
(********************************************************************
 * COPYRIGHT -- Herbert Kannegiesser GmbH
 ********************************************************************
 * Library: KanLinkLib
 * File: KLLib_CfgServer.st
 * Author: stahlhut
 * Created: February 01, 2012
 ********************************************************************
 * Implementation of library KanLinkLib
 ********************************************************************)

(* Configuriert einen Kanlink Server *)
FUNCTION_BLOCK KLLib_CfgServer
	// überprüfen
	IF (adrKanlink = 0) OR (adrSReq = 0) OR (adrSResp = 0) OR (adrName = 0)  THEN
		status := 1; // Fehler 1 adressen fehler
		RETURN;
	END_IF;
	IF (ServerIndex > HLKANLINK_MAX_SERVERCONNS) THEN
		status := 2; // Fehler Index zu gross
		RETURN;
	END_IF;

	_dKL ACCESS adrKanlink;
	IF _dKL.ServerListe[ServerIndex].adrParameter = 0 THEN
		status := 3; // fehler Kanlink / fehlende init der adressen Interface
		RETURN;
	END_IF;

	IF TimeOut < 200 THEN
		TimeOut := 1000;
	END_IF;

	_dSrvPar ACCESS _dKL.ServerListe[ServerIndex].adrParameter;
	_dSrvPar.Adr := IPAdr;
	_dSrvPar.Area := Area;
	_dSrvPar.Cmd := Cmd;
	_dSrvPar.CmdOpt := CmdOpt;
	memcpy(ADR( _dSrvPar.Name ),adrName,15);
	memcpy(ADR(_dSrvPar.sReq),adrSReq,80);
	memcpy(ADR(_dSrvPar.sResp),adrSResp,80);
	_dSrvPar.TimeOut := TimeOut;

	_iret := KLLib_ReadServerPara(ADR(_dKL.ServerListe[ServerIndex]),(_dKL.ServerListe[ServerIndex].adrParameter));

	IF ( _iret <> 0 ) THEN
		status := 4;
	ELSE
		status := 0; // mit ok beenden
	END_IF;

END_FUNCTION_BLOCK
```

#### KanLink_FB.st
```iecst
(********************************************************************
 * COPYRIGHT -- Herbert Kannegiesser GmbH
 ********************************************************************
 * Library: WetLinkLib
 * File: WL_Data.st
 * Author: stahlhut
 * Created: January 06, 2012
 ********************************************************************
 * Implementation of library WetLinkLib
 ********************************************************************)

(* TODO: Add your comment here *)
FUNCTION_BLOCK KanLink_FB

	xReturn := 0;

	IF Step <> 10 THEN
		xReturn := 1;
		RETURN;
	END_IF;
	KLLib_ClientTimer(adrSelf,_iCycleTime);

	IF UdpSend_0.enable THEN
		UdpSend_0;
		IF UdpSend_0.status = 0 THEN
			UdpSend_0.enable := FALSE;
		ELSIF UdpSend_0.status = ERR_FUB_BUSY THEN
			UdpSend_0.enable := TRUE;

			xReturn := 1;
			RETURN;
		ELSE
			ErrorNr := 4;

//			IF_WLLogger.Logitem.error_number := WL_ErrorNr;
//			IF_WLLogger.Logitem.binary_data := Server.UdpSend_0.status;
//			IF_WLLogger.Logitem.loglevel := 3;
//			IF_WLLogger.Logitem.ascii_data := 'WL unable to send data';
//			IF_WLLogger.xStart := TRUE;
			UdpSend_0.enable := FALSE;
		END_IF
	END_IF;

	UdpRecv_0.enable := 1;
	UdpRecv_0.ident := UdpOpen_0.ident;
	UdpRecv_0.pData := ADR(ServerData.receive_data);	// Datenspeicher
	UdpRecv_0.datamax := SIZEOF(ServerData.receive_data);	// Länge des Datenspeichers
	UdpRecv_0.flags := 0;
	UdpRecv_0.pIpAddr := ADR(client_address);	// IP Adresse des Senders
	UdpRecv_0;

	IF UdpRecv_0.status = 0 THEN  // Daten empfangen
		// Header Daten kopieren

		_dPrehead ACCESS ADR(ServerData.receive_data);
		_dHead ACCESS ADR(ServerData.receive_data) + PreHeaderSize;
		memcpy(ADR(ServerData.PreHeaderRec),ADR(ServerData.receive_data),PreHeaderSize);
		memcpy(ADR(ServerData.HeaderV1Rec),ADR(ServerData.receive_data)+PreHeaderSize,SIZEOF(ServerData.HeaderV1Rec));

		ethInetAton(ADR(client_address),ADR(_dRecAdr));
		_udArr ACCESS ADR(_dRecAdr);

		ServerData.recArea := _udArr.c;
		ServerData.recAddr := _udArr.d;

		_xPreheadOK := (ServerData.PreHeaderRec.Magic = MagicNr);
		_xVersionOK := (ServerData.PreHeaderRec.HeaderVersion = 16#100);

		IF (_dHead.Command AND 1) = 0 THEN
			_xGetServerReq := TRUE;
		ELSIF (_dHead.Command AND 1) = 1 THEN
			_xGetClientResp := TRUE;
		END_IF;

	ELSIF UdpRecv_0.status = udpERR_NO_DATA THEN  // Keine Daten empfangen, Client abarbeiten
		_xSendClient := TRUE;
	ELSIF UdpRecv_0.status = ERR_FUB_BUSY THEN  (* UdpRecv not finished -> redo *)
		xReturn := 1;
		RETURN;
	ELSE  (* Goto Error Step *)
		ErrorNr := 5;
//		IF_WLLogger.Logitem.error_number := WL_ErrorNr;
//		IF_WLLogger.Logitem.binary_data := Server.UdpRecv_0.status;
//		IF_WLLogger.Logitem.loglevel := 3;
//		IF_WLLogger.Logitem.ascii_data := 'WL unable to receive data';
//		IF_WLLogger.xStart := TRUE;
		xReturn := 1;
		RETURN;
	END_IF

END_FUNCTION_BLOCK
```

#### KLLib_ClientTimer.st
```iecst
(********************************************************************
 * COPYRIGHT -- Herbert Kannegiesser GmbH
 ********************************************************************
 * Library: WetLinkLib
 * File: WLLIb_ClientTimer.st
 * Author: stahlhut
 * Created: January 06, 2012
 ********************************************************************
 * Implementation of library WetLinkLib
 ********************************************************************)

(* TODO: Add your comment here *)
FUNCTION KLLib_ClientTimer
FOR _i := 0 TO HLKANLINK_MAX_CLIENTCONNS DO
	_dClient  ACCESS ADR(Srv.ClientListe[_i]);
	_dInterface ACCESS (_dClient.adrInterface);

	// TimeOut (kurz) taskgerecht berechnen
	IF (_dClient.TimeOutLeft >= _iCycleTime) AND _dClient.xReqPending THEN
 		_dClient.TimeOutLeft := _dClient.TimeOutLeft - _iCycleTime;
	END_IF;

	IF _dClient.iCycleWait <= _dClient.iCycleTime THEN
		_dClient.iCycleWait := _dClient.iCycleWait + _iCycleTime;
	END_IF;
	// Timeout aufgetreten nur bis n Zählen. Retry sofort nach timeout, sonst retry nach cycletime
	IF _dClient.xReqPending AND (_dClient.TimeOutLeft < _iCycleTime) THEN
		_dClient.iTimeOutCnt_Summe := _dClient.iTimeOutCnt_Summe + 1;
		_dClient.xReqPending := FALSE;	// noch mal versuchen
		IF _dClient.iTimeOutCnt < 5 THEN
			_dClient.iTimeOutCnt := _dClient.iTimeOutCnt +1 ;
			_dClient.xReqPending := FALSE;	// noch mal versuchen
			_dInterface.iState := 4;
			_dClient.iCycleWait := _dClient.iCycleTime;
		END_IF;
	END_IF;
		// Verbindungsfehler
	_dClient.xConnected := (_dClient.iTimeOutCnt < 5) AND _dClient.xActiv AND (_dClient.iCycleTime > 0);
	_dInterface.out.xConnected := _dClient.xConnected;
	IF (_dClient.iTimeOutCnt >= 5 ) AND ( _dInterface.iState = 2 ) THEN
		_dInterface.iState := 255; // Timeout melden
	END_IF;

END_FOR;

FOR _i := 0 TO HLKANLINK_MAX_SERVERCONNS DO
	_dServer ACCESS ADR(Srv.ServerListe[_i]);
	_dSrvIf ACCESS _dServer.adrInterface;

	IF _dServer.iConnectionTimer <= 2000 THEN
		_dServer.iConnectionTimer := _dServer.iConnectionTimer + _iCycleTime;
	END_IF;
	_dServer.xConnected := (_dServer.iConnectionTimer < 2000);
	_dSrvIf.out.xConnected := _dServer.xConnected;

END_FOR;

END_FUNCTION
```

#### KLLib_GetPVAdr.st
```iecst
(********************************************************************
 * COPYRIGHT -- Herbert Kannegiesser GmbH
 ********************************************************************
 * Library: WetLinkLib
 * File: WLLib_GetPVAdr.st
 * Author: stahlhut
 * Created: January 06, 2012
 ********************************************************************
 * Implementation of library WetLinkLib
 ********************************************************************)

(* TODO: Add your comment here *)
FUNCTION KLLib_GetPVAdr
	iStat := PV_xgetadr((ServerItem.pReqStr),ADR(ServerItem.AdrDataReq),ADR(ServerItem.ReqLength));
	IF iStat <> 0 THEN // fehler aufgetreten
 		ServerItem.AdrDataReq := 0;
		ServerItem.ReqLength := 0;
	END_IF;
	iStat := PV_xgetadr((ServerItem.pRespStr),ADR(ServerItem.AdrDataResp),ADR(ServerItem.RespLength));
	IF iStat <> 0 THEN // fehler aufgetreten
 		ServerItem.AdrDataResp := 0;
		ServerItem.RespLength := 0;
	END_IF;

END_FUNCTION
```

#### KLLib_SendData.st
```iecst
(********************************************************************
 * COPYRIGHT -- Herbert Kannegiesser GmbH
 ********************************************************************
 * Library: WetLinkLib
 * File: WLLib_SendData.st
 * Author: stahlhut
 * Created: January 07, 2012
 ********************************************************************
 * Implementation of library WetLinkLib
 ********************************************************************)

(* TODO: Add your comment here *)
FUNCTION KLLib_SendData
	IF Srv.UdpSend_0.enable = TRUE THEN //Sendung noch unterwegs, abbrechen
 		KLLib_SendData := 1;
		RETURN;
	END_IF;

	Srv.ServerData.PreHeaderSend.Magic := MagicNr;
	Srv.ServerData.PreHeaderSend.HeaderVersion := 16#0100;
	Srv._offset := 0;
	memcpy(ADR(Srv.ServerData.send_data),ADR(Srv.ServerData.PreHeaderSend),PreHeaderSize);
	Srv._offset := PreHeaderSize;

	memcpy(ADR(Srv.ServerData.send_data)+Srv._offset,ADR(Srv.ServerData.HeaderV1Send),HeaderSize);
	Srv._offset := Srv._offset+ HeaderSize;
	memcpy(ADR(Srv.ServerData.send_data)+Srv._offset,SendAdr,SendLen);
	Srv._SendLen := Srv._offset + Srv.ServerData.HeaderV1Send.Length;

	// Telegramm jetzt senden
	Srv.UdpSend_0.enable := 1;
	Srv.UdpSend_0.ident 	:= Srv.UdpOpen_0.ident;	(* Client Ident from AsUDP.UDP_Open *)
	Srv.UdpSend_0.pHost 	:= pDestination;	(* IP Address of the Client *)
	Srv.UdpSend_0.port 	:= Srv.iPort;
	Srv.UdpSend_0.pData 	:= ADR(Srv.ServerData.send_data);	(* Which data to send *)
	Srv.UdpSend_0.datalen :=  Srv._SendLen; //
	Srv.UdpSend_0.flags 	:= 0;
	Srv.UdpSend_0 ;	(* Call the Function*)

END_FUNCTION
```

#### KLLib_ReadServerPara.st
```iecst
(********************************************************************
 * COPYRIGHT -- Herbert Kannegiesser GmbH
 ********************************************************************
 * Library: WetLinkLib
 * File: WLLib_ReadServerPara.st
 * Author: stahlhut
 * Created: January 08, 2012
 ********************************************************************
 * Implementation of library WetLinkLib
 ********************************************************************)

(* TODO: Add your comment here *)
FUNCTION KLLib_ReadServerPara

_xError := (adrServerItem = 0) OR (adrParaItem=0);

IF _xError THEN // Fehler aufgetreten
	dServer.iCfgStatus := 2;
	KLLib_ReadServerPara := 1;
ELSE
	dServer ACCESS adrServerItem;
	dPara ACCESS adrParaItem;

	dServer.iCfgStatus := 0;

	dServer.Cmd :=  dPara.Cmd;
	dServer.CmdOpt := dPara.CmdOpt;
	dServer.Adr :=  dPara.Adr;
	dServer.Area := dPara.Area;
	dServer.pReqStr := ADR(dPara.sReq);
	dServer.pRespStr := ADR(dPara.sResp);
	dServer.adrParameter := adrParaItem;
	dServer.xReqManually := (dPara.CmdOpt AND KL_optReqManually) <> 0 ;
	KLLib_ReadServerPara := 0;

	dServer.Key := KL_BuildKey(Command:= (dServer.Cmd),CmdNr := UINT_TO_USINT( dPara.CmdOpt) ,Area := UINT_TO_USINT( dPara.Area ),IPAdr := UINT_TO_USINT( dPara.Adr));
	KLLib_GetPVAdr(adrServerItem);
	IF (dServer.AdrDataReq= 0) OR (dServer.AdrDataResp = 0) THEN
		dServer.iCfgStatus := 1; // fehler melden
	END_IF;
END_IF;

END_FUNCTION
```

#### KLLib_ReadClientPara.st
```iecst
(********************************************************************
 * COPYRIGHT -- Herbert Kannegiesser GmbH
 ********************************************************************
 * Library: WetLinkLib
 * File: WLLib_ReadClientPara.st
 * Author: stahlhut
 * Created: January 08, 2012
 ********************************************************************
 * Implementation of library WetLinkLib
 ********************************************************************)

(* TODO: Add your comment here *)
FUNCTION KLLib_ReadClientPara
_xError := (adrClientItem = 0) OR (adrParaItem=0) OR (adrServer = 0);

IF _xError THEN // Fehler aufgetreten
	KLLib_ReadClientPara := 1;
ELSE
	dClient ACCESS adrClientItem;
	dPara ACCESS adrParaItem;
	dServer ACCESS adrServer;
	dClient.Cmd :=  dPara.Cmd;
	dClient.RecCmd := dPara.Cmd + 1 ;
	dClient.Adr :=  dPara.Adr;
	dClient.Area := dPara.Area;
	dClient.iCycleTime := dPara.CycleTime;
	dClient.pReq := ADR(dPara.sReq);
	dClient.pResp := ADR(dPara.sResp);
	dClient.adrParameter := adrParaItem;
	dClient.CmdOpt := dPara.CmdOpt;
	KLLib_ReadClientPara := 0;

	KLLib_InitCltPV(adrClientItem);
	 dClient.Key := KL_BuildKey(Command:= dClient.RecCmd,CmdNr:=  UINT_TO_USINT( dPara.CmdOpt),Area := UINT_TO_USINT( dPara.Area), IPAdr := UINT_TO_USINT( dPara.Adr));

	// Host string erzeugen

	_udArr ACCESS ADR(_udAdr );
	_udNetId ACCESS ADR(dServer.udNetID);
	_udArr.a := _udNetId.a;
	_udArr.b := _udNetId.b;
	_udArr.c := (_udNetId.c AND 16#F0) +  UINT_TO_USINT( dClient.Area);
	_udArr.d := UINT_TO_USINT( dClient.Adr);

	ethInetNtoa((_udAdr),ADR(dClient.sClientAdr));

END_IF;

END_FUNCTION
```

#### KL_BuildKey.st - Berechnen des Connection Key
```iecst
(********************************************************************
 * COPYRIGHT -- Herbert Kannegiesser GmbH
 ********************************************************************
 * Library: KanLinkLib
 * Datei: KL_BuildKey.st
 * Autor: stahlhut
 * Erstellt: 16. Januar 2012
 ********************************************************************
 * Implementierung der Library KanLinkLib
 ********************************************************************)

(* Berechnen des Connection Key *)
FUNCTION KL_BuildKey

	KL_BuildKey := SHL(UINT_TO_UDINT(Command),16)+SHL(USINT_TO_UINT(CmdNr),12)+SHL(USINT_TO_UINT(Area),8)+ (IPAdr AND 16#00FF);

END_FUNCTION
```

#### KLLib_Init.st
```iecst
(********************************************************************
 * COPYRIGHT -- Herbert Kannegiesser GmbH
 ********************************************************************
 * Library: KanLinkLib
 * File: KL_Init.st
 * Author: stahlhut
 * Created: January 12, 2012
 ********************************************************************
 * Implementation of library KanLinkLib
 ********************************************************************)

(* TODO: Add your comment here *)
FUNCTION_BLOCK KLLib_Init

	IF (adrServer = 0) OR (adrInterface = 0 )  THEN // fehler
		status := 1;
		enable := 0;
		RETURN;
	END_IF;
	IF enable = 0 THEN
		status := ERR_FUB_ENABLE_FALSE;
		RETURN;
	END_IF;

	IF (status = ERR_FUB_BUSY	) AND (enable = 0) THEN
		status := ERR_FUB_ENABLE_FALSE;
		_bStep := 100;
	END_IF;

	CASE _bStep OF
		0: // nix tun
			status := ERR_FUB_BUSY;
			_bStep := 10;
		10:
			_dServer ACCESS adrServer;
			_dServer.adrSelf := adrServer;
			_dIf ACCESS adrInterface;
			_dServer.adrInterface := adrInterface;

			IF _dServer.iPort = 0 THEN
				_dServer.iPort := 23500; // standardport benutzen
			END_IF;
			RTInfo_0.enable := TRUE;
			RTInfo_0;

			_dServer._iCycleTime := UDINT_TO_UINT( RTInfo_0.cycle_time / 1000);

			_bStep := 20;
		20:
			GetEthPort_0.enable := 1;
			GetEthPort_0.adrIF := ADR(_dServer.sIF);
			GetEthPort_0;
			IF GetEthPort_0.status = ERR_OK THEN
				_bStep := 30;
			ELSIF GetEthPort_0.status <> ERR_FUB_BUSY THEN // fehler aufgetreten
				status := 2;
				_bStep := 100;
			END_IF;
		30:
			CfgGetIPAddr_0.enable  := 1;
			CfgGetIPAddr_0.pDevice := ADR(_dServer.sIF);
			CfgGetIPAddr_0.pIPAddr := ADR(_dServer.sNetID);
			CfgGetIPAddr_0.Len := 16;
			CfgGetIPAddr_0;
			IF  (CfgGetIPAddr_0.status = ERR_OK) THEN
				_bStep := 40;
				ethInetAton(ADR(_dServer.sNetID),ADR(_dServer.udNetID));

			ELSIF CfgGetIPAddr_0.status <> ERR_FUB_BUSY THEN // fehler aufgetreten
				status := 3;
				_bStep := 100;
			END_IF;

		40:
			FOR _i := 0 TO HLKANLINK_MAX_SERVERCONNS DO
				_dServer.ServerListe[_i].adrInterface := ADR(_dIf.Server[_i]);
				KLLib_ReadServerPara(ADR(_dServer.ServerListe[_i]), ADR( _dIf.Parameter.Server[_i]));
			END_FOR;
			//			memset(ADR(_dServer.ClientListe),0,SIZEOF(_dServer.ClientListe));
			FOR _i := 0 TO HLKANLINK_MAX_CLIENTCONNS DO
				KLLib_ReadClientPara(ADR(_dServer.ClientListe[_i]),ADR(_dIf.Parameter.Client[_i]),ADR(_dServer));
				_dServer.ClientListe[_i].xActiv := (_dServer.ClientListe[_i].Cmd <> 0);
				_dServer.ClientListe[_i].TimeOut := 140;
				_dServer.ClientListe[_i].adrInterface := ADR(_dIf.Client[_i]);
			END_FOR;
			_bStep := 50;
		50:

			_dServer.UdpOpen_0.enable := 1;
			_dServer.UdpOpen_0.pIfAddr := 0;//ADR(Server.sIF);	(* Übergeben des Interface funzt nicht *)
			_dServer.UdpOpen_0.port := _dServer.iPort;	(* Port to listen*)
			_dServer.UdpOpen_0.options := 0;
			_dServer.UdpOpen_0;	(* Call the Function*)

			IF _dServer.UdpOpen_0.status = 0 THEN  (* UdpOpen successful*)
				_dServer._uiLastId := _dServer.UdpOpen_0.ident;
				_bStep := 90;
			ELSIF _dServer.UdpOpen_0.status = ERR_FUB_BUSY THEN  (* UdpOpen not finished -> redo *)

			ELSIF _dServer.UdpOpen_0.status = udpERR_ALREADY_EXIST THEN // erst schliessen
				_dServer.UdpClose_0.enable := 1;
				_dServer.UdpClose_0.ident := _dServer._uiLastId;
				_dServer.UdpClose_0;
				IF _dServer.UdpClose_0.status = 0 THEN
					//
				ELSIF _dServer.UdpClose_0.status = ERR_FUB_BUSY THEN

				ELSE
					status := 5001;
					_bStep := 100;	// unbekannter close fehler aufgetreten
				END_IF;

			ELSE
				status := 5002;
				_bStep := 100; // unbekannter open fehler aufgetreten
			END_IF

//			_dServer.DoCommand := 10;
//			_dServer;
//			IF _dServer.DoCommand = 0 THEN // Ausgeführt weiter
//				_bStep := 90;
//				_dServer.UdpRecv_0.enable := 1;
//			ELSIF _dServer.DoCommand = 1000 THEN // fehler aufgetreten
//				status := 4;
//				_bStep := 100;
////				IF_WLLogger.Logitem.error_number := WL_ErrorNr;
////				IF_WLLogger.Logitem.binary_data := (Server.UdpOpen_0.status);
////				IF_WLLogger.Logitem.loglevel := 3;
////				IF_WLLogger.Logitem.ascii_data := 'WL unable to open Port ';
////				IF_WLLogger.xStart := TRUE;
//
//			END_IF;

		90:  // fertig
			status := ERR_OK;
			enable := 0;
			_bStep := 0;

		100: // fehler aufgetreten
			enable := 0;
			_bStep := 0;

	END_CASE;

END_FUNCTION_BLOCK
```

#### KLLib_CreateStrucDef.st - Erzeuge eine Strukturdefinition zu einer Variablen
```iecst
(********************************************************************
 * COPYRIGHT -- Herbert Kannegiesser GmbH
 ********************************************************************
 * Library: KanLinkLib
 * File: KLLib_CreateStrucDef.st
 * Author: hunholz
 * Created: February 23, 2012
 ********************************************************************
 * Implementation of library KanLinkLib
 ********************************************************************)

(* Erzeuge eine Strukturdefinition zu einer Variablen *)

(* 1. Array müssen bei 0 beginnen
   2. Enumerationen und abgeleitete Datentypen sind verboten
*)
FUNCTION KLLib_CreateStrucDef

	KLLib_CreateStrucDef := ERR_OK;

	IF lPtrAdr = 0 OR lPtrLen = 0 THEN

		KLLib_CreateStrucDef := KLLIB_MSG_NULL_POINTER;
		RETURN;

	END_IF

	_sPvName := sRootName;

	_lAdr ACCESS lPtrAdr;
	_lLen ACCESS lPtrLen;

	IF _lAdr = 0 THEN
		KLLib_CreateStrucDef := KLLIB_MSG_NULL_POINTER;
		RETURN;
	END_IF

	IF sItemName <> '' THEN
		_sPvName := CONCAT(_sPvName, '.');
		_sPvName := CONCAT(_sPvName, sItemName);
	ELSE
		brsmemset(_lAdr, 0, _lLen);
	END_IF

	_wStatus := PV_ninfo(ADR(_sPvName), ADR(_lDataType), ADR(_lDataLen), ADR(_wDataDimension));

	IF _wStatus = ERR_OK THEN

		_sValueDim := UINT_TO_STRING(_wDataDimension);
		_sValueLen := UDINT_TO_STRING(_lDataLen);

		_wStatus := PV_xgetadr(ADR(_sPvName), ADR(_lDataAdr), ADR(_lDataLen));

		IF lDataAdr > 0 AND _lDataAdr > lDataAdr THEN

			_sValueOffs := UDINT_TO_STRING(_lDataAdr - lDataAdr);

		ELSE

			_sValueOffs := '0';

		END_IF

		CASE _lDataType OF

			0:  // Struktur

				_sLine := 'STRUC$T';
				_sLine := CONCAT(_sLine, sItemName);
				_sLine := CONCAT(_sLine, '$T');
				_sLine := CONCAT(_sLine, _sValueLen);
				_sLine := CONCAT(_sLine, '$T');
				_sLine := CONCAT(_sLine, _sValueOffs);
				_sLine := CONCAT(_sLine, '$T1');

				_wStatus := KLLib_WriteStrucDefLine(lPtrLine := ADR(_sLine), lPtrAdr := lPtrAdr, lPtrLen := lPtrLen);

				IF _wStatus <> ERR_OK THEN

					KLLib_CreateStrucDef := _wStatus;
					RETURN;

				END_IF

				// Die einzelnen Elemente der Struktur ermitteln

				FOR _i := 1 TO _wDataDimension DO

					_wStatus := PV_item(ADR(_sPvName), _i-1, ADR(_sItemName));

					IF _wStatus = ERR_OK THEN

						// Rekursion mit dem Strukturelement

						_wStatus := KLLib_CreateStrucDef(lPtrAdr := lPtrAdr, lPtrLen := lPtrLen, sRootName := _sPvName, sItemName := _sItemName, lDataAdr := _lDataAdr);

						IF _wStatus <> ERR_OK THEN
							KLLib_CreateStrucDef := _wStatus;
							RETURN;
						END_IF

					ELSE
						KLLib_CreateStrucDef := _wStatus;
						RETURN;
					END_IF

				END_FOR

				_sLine := 'ENDSTRUC';

				_wStatus := KLLib_WriteStrucDefLine(lPtrLine := ADR(_sLine), lPtrAdr := lPtrAdr, lPtrLen := lPtrLen);

				IF _wStatus <> ERR_OK THEN

					KLLib_CreateStrucDef := _wStatus;
					RETURN;

				END_IF

			15:	// Array einer Struktur

				_sLine := 'STRUC$T';
				_sLine := CONCAT(_sLine, sItemName);
				_sLine := CONCAT(_sLine, '$T');
				_sLine := CONCAT(_sLine, _sValueLen);
				_sLine := CONCAT(_sLine, '$T');
				_sLine := CONCAT(_sLine, _sValueOffs);
				_sLine := CONCAT(_sLine, '$T');
				_sLine := CONCAT(_sLine, _sValueDim);

				_wStatus := KLLib_WriteStrucDefLine(lPtrLine := ADR(_sLine), lPtrAdr := lPtrAdr, lPtrLen := lPtrLen);

				IF _wStatus <> ERR_OK THEN

					KLLib_CreateStrucDef := _wStatus;
					RETURN;

				END_IF

				// Um die Elemente der Struktur zu ermitteln wird PV_ninfo erneut mit einem Element des Array aufgerufen

				_sPvName := CONCAT(_sPvName,'[0]');

				_wStatus := PV_ninfo(ADR(_sPvName), ADR(_lDataType), ADR(_lDataLen), ADR(_wDataDimension));

				IF _wStatus = ERR_OK THEN

					// Die einzelnen Elemente der Struktur ermitteln

					FOR _i := 1 TO _wDataDimension DO

						_wStatus := PV_item(ADR(_sPvName), _i-1, ADR(_sItemName));

						IF _wStatus = ERR_OK THEN

							// Rekursion mit dem Strukturelement

							_wStatus := KLLib_CreateStrucDef(lPtrAdr := lPtrAdr, lPtrLen := lPtrLen, sRootName := _sPvName, sItemName := _sItemName, lDataAdr := _lDataAdr);

							IF _wStatus <> ERR_OK THEN
								KLLib_CreateStrucDef := _wStatus;
								RETURN;
							END_IF

						ELSE
							KLLib_CreateStrucDef := _wStatus;
							RETURN;
						END_IF

					END_FOR

					_sLine := 'ENDSTRUC';

					_wStatus := KLLib_WriteStrucDefLine(lPtrLine := ADR(_sLine), lPtrAdr := lPtrAdr, lPtrLen := lPtrLen);

					IF _wStatus <> ERR_OK THEN

						KLLib_CreateStrucDef := _wStatus;
						RETURN;

					END_IF

				ELSE

					KLLib_CreateStrucDef := KLLIB_MSG_VAR_ERROR;
					RETURN;

				END_IF

			1..14,16..23:

				_sLine := CONCAT(_sType[_lDataType],'$T');
				_sLine := CONCAT(_sLine, sItemName);
				_sLine := CONCAT(_sLine, '$T');
				_sLine := CONCAT(_sLine, _sValueLen);
				_sLine := CONCAT(_sLine, '$T');
				_sLine := CONCAT(_sLine, _sValueOffs);
				_sLine := CONCAT(_sLine, '$T');
				_sLine := CONCAT(_sLine, _sValueDim);

				_wStatus := KLLib_WriteStrucDefLine(lPtrLine := ADR(_sLine), lPtrAdr := lPtrAdr, lPtrLen := lPtrLen);

				IF _wStatus <> ERR_OK THEN

					KLLib_CreateStrucDef := _wStatus;
					RETURN;

				END_IF

		END_CASE

	ELSE

		KLLib_CreateStrucDef := _wStatus;
		RETURN;

	END_IF

END_FUNCTION
```

#### KLLib_WriteStrucDefLine.st - Übertrage einen String als Zeile in den Speicher
```iecst
(********************************************************************
 * COPYRIGHT -- Herbert Kannegiesser GmbH
 ********************************************************************
 * Library: KanLinkLib
 * File: KLLib_WriteStrucDefLine.st
 * Author: hunholz
 * Created: February 24, 2012
 ********************************************************************
 * Implementation of library KanLinkLib
 ********************************************************************)

(* Übertrage einen String als Zeile in den Speicher *)
FUNCTION KLLib_WriteStrucDefLine

	IF lPtrAdr = 0 OR lPtrLen = 0 OR lPtrLine = 0 THEN

		KLLib_WriteStrucDefLine := KLLIB_MSG_NULL_POINTER;
		RETURN;

	END_IF

	_lAdr ACCESS lPtrAdr;
	_lLen ACCESS lPtrLen;
	_sLine ACCESS lPtrLine;

	_sLine := CONCAT(_sLine, '$R$L');

	_iStringlen := LEN(_sLine);

	IF (_iStringlen+1) > _lLen THEN

		KLLib_WriteStrucDefLine := KLLIB_MSG_NOT_ENOUGH_MEM;
		RETURN;

	ELSE

		brsstrcpy(_lAdr, lPtrLine);
		_lAdr := _lAdr + INT_TO_UDINT(_iStringlen);
		_lLen := _lLen - INT_TO_UDINT(_iStringlen);

	END_IF

	KLLib_WriteStrucDefLine := ERR_OK;

END_FUNCTION
```

### history.txt
```
21.02.12 sta 0.93
Client kann mit state gesteuert werden

8.2.12 sta 0.92
Fehler bei Server-Key behoben
2.2.12 sta
Zum einrichten eines Server und Client KLLib_CfgServer und KLLib_CfgClient integriert.
Konf sowohl über Parameter und mit den Funktionen möglich

30.1.12 sta
interface  umbenannt
MaxServerConn und MaxClientCon in userlib

todo:
"OneShot" Client-Statevariable
Überprüfung Längen der Commandos
Logger wieder inbetriebnehmen

Startversion 0.900
```

### Package Logical/Mewa/KGFramework/Pkg_mnTest - Testadapter für automatische Tests

### Pkg_mnTest.var - Package variables
```iecst
(********************************************************************
 * COPYRIGHT -- Herbert Kannegiesser GmbH
 ********************************************************************
 * Package: Pkg_mnTest
 * File: Pkg_mnTest.var
 * Author: hunholz
 * Created: March 06, 2012
 ********************************************************************
 * Variables of package Pkg_mnTest
 ********************************************************************)
VAR
	IFmnTest : IFmnTest_typ;
	mnTestCmd : KG_Cmd_typ;
	mnTestStatAd : mnTestStatAd_typ;
	mnTestStat : Stat_typ;
END_VAR
(*KONSTANTEN*)
VAR CONSTANT
	MNTEST_CMD_SETMODE : UINT := 1000; (*Mode steht in lData0*)
	MNTEST_CMD_RESET : UINT := 1001; (*Warm- oder Kaltstart, siehe lData0*)
	MNTEST_CMDSTAT_SETMODEFAILED : UINT := 60000;
	MNTEST_TESTMODE_INTERFACE : UINT := 1; (*Reiner Interfacetest*)
	MNTEST_TESTMODE_MAX : UINT := 1;
	MNTEST_RESETMODE_WARMSTART : USINT := 1;
	MNTEST_RESETMODE_COLDSTART : USINT := 2;
	MNTEST_STAT_ERRFBSETMODE : UINT := 60000; (*Fehler aus _fbSetMode. Siehe sStatus*)
	MNTEST_STAT_ERRMSGCFGCNT : UINT := 60001; (*Falsche Anzahl Meldungen*)
	MNTEST_STAT_ERRMSGCFG : UINT := 60002; (*Fehler DatObjInfo*)
	MNTEST_STAT_FBRUNTEST : UINT := 60003; (*Fehler aus _fbRunTest. Siehe sStatus*)
END_VAR
```

### Program Logical/Mewa/KGFramework/Pkg_mnTest/mnTest (IEC) - Testadapter

#### mnTestCyclic.st - Cyclic code
```iecst
(********************************************************************
 * COPYRIGHT -- Herbert Kannegiesser GmbH
 ********************************************************************
 * Program: mnTest
 * File: mnTestCyclic.st
 * Author: hunholz
 * Created: March 03, 2012
 ********************************************************************
 * Implementation of program mnTest
 ********************************************************************)

PROGRAM _CYCLIC

	//====================
	// Kommandointerpreter
	//====================

	CASE _CommandoState OF

		_csIdle:

			CASE mnTestCmd.Request.Command.wCommand OF

				KG_CMD_NOCOMMAND:

					mnTestCmd.Response.wCmdStatus := KG_CMD_NOCOMMAND;

				MNTEST_CMD_RESET:

					IF mnTestCmd.Request.Command.lData0 <> MNTEST_RESETMODE_WARMSTART AND mnTestCmd.Request.Command.lData0 <> MNTEST_RESETMODE_COLDSTART THEN

						mnTestCmd.Response.wCmdStatus := KG_CMDSTAT_INVALID_PARAMETER;

					ELSE

						SYSreset(enable := TRUE, mode := UDINT_TO_USINT(mnTestCmd.Request.Command.lData0));
						mnTestCmd.Response.wCmdStatus := MNTEST_CMD_RESET;

					END_IF

					_CommandoState := _csWaitForNull;

				MNTEST_CMD_SETMODE:

					IF _wTestMode <> 0 THEN

						mnTestCmd.Response.wCmdStatus := MNTEST_CMDSTAT_SETMODEFAILED;

					ELSIF mnTestCmd.Request.Command.lData0 = 0 OR mnTestCmd.Request.Command.lData0 > MNTEST_TESTMODE_MAX THEN

						mnTestCmd.Response.wCmdStatus := KG_CMDSTAT_INVALID_PARAMETER;

					ELSE

						_wTestMode := UDINT_TO_UINT(mnTestCmd.Request.Command.lData0);
						mnTestCmd.Response.wCmdStatus := MNTEST_CMD_SETMODE;
						_TestState := _tsSetMode;

					END_IF

					_CommandoState := _csWaitForNull;

				ELSE

					_CommandoState := _csWaitForNull;
					mnTestCmd.Response.wCmdStatus := KG_CMDSTAT_NOTVALID;

			END_CASE

		_csWaitForNull:

			IF mnTestCmd.Request.Command.wCommand = KG_CMD_NOCOMMAND THEN

				_CommandoState := _csIdle;
				mnTestCmd.Response.wCmdStatus := KG_CMD_NOCOMMAND;

			END_IF

		ELSE

			_CommandoState := _csIdle;

	END_CASE

	//======================
	// Statemachine Testmode
	//======================

	CASE _TestState OF

		_tsIdle:

			// Tue nichts

		_tsSetMode:

			_fbSetMode(enable := TRUE, pStruc := IFmnTest.In.pStrucTest, wMode := _wTestMode);

			IF _fbSetMode.status = ERR_OK THEN

				// Framework darf keine Meldungen mehr erzeugen und das
				// Meldesystem wird zurückgesetzt
				IFmnTest.Out.xNoMessages := TRUE;
				brsmemset(ADR(kgMsgStatus),0,SIZEOF(kgMsgStatus));

				_TestState := _tsPrepTest1;

			ELSE

				_TestState := _tsFault;

				mnTestStat.wStatus := MNTEST_STAT_ERRFBSETMODE;
				mnTestStat.sStatus := UINT_TO_STRING(_fbSetMode.status);

			END_IF

		_tsPrepTest1:

			_doInfoCfg.enable := TRUE;	// VAR_INPUT BOOL enable 'enables execution'
			_doInfoCfg.pName := ADR('CfgMsgStat');	// VAR_INPUT UDINT pName 'name of data object'
			_doInfoCfg();

			IF _doInfoCfg.status = ERR_OK THEN

				_wMsgCnt := UDINT_TO_UINT((_doInfoCfg.len-SIZEOF(UINT))/SIZEOF (MsgCfgLine_Typ)); // Laenge der Version zu Beginn abziehen

				IF _wMsgCnt > 0 AND _wMsgCnt <= MNMSG_MAX_CFGMESSAGES THEN

					_MsgCfgList ACCESS _doInfoCfg.pDatObjMem + SIZEOF(UINT);
					_TestState := _tsRun;

				ELSE
					// Meldungskonfiguration fehlerhaft
					_TestState := _tsFault;

					mnTestStat.wStatus := MNTEST_STAT_ERRMSGCFGCNT;
					mnTestStat.sStatus := UINT_TO_STRING(_wMsgCnt);

				END_IF

			ELSE
				// Meldungskonfiguration fehlt
				_TestState := _tsFault;
				mnTestStat.wStatus := MNTEST_STAT_ERRMSGCFG;
				mnTestStat.sStatus := UINT_TO_STRING(_doInfoCfg.status);

			END_IF

		_tsRun:

			_fbRunTest(enable := TRUE, pStruc := IFmnTest.In.pStrucTest, wMode := _wTestMode);

			IF _fbRunTest.status <> ERR_OK THEN

				_TestState := _tsFault;

				mnTestStat.wStatus := MNTEST_STAT_FBRUNTEST;
				mnTestStat.sStatus := UINT_TO_STRING(_fbRunTest.status);

			END_IF

			// ACTION RUN MessageTest
			_MessageTest1;

		_tsFault:

			// Tue erstmal nichts

	END_CASE

END_PROGRAM
```

#### mnTest.var - Local variables
```iecst
(********************************************************************
 * COPYRIGHT -- Herbert Kannegiesser GmbH
 ********************************************************************
 * Program: mnTest
 * File: mnTest.var
 * Author: hunholz
 * Created: March 03, 2012
 ********************************************************************
 * Local variables of program mnTest
 ********************************************************************)
(*Packageversion auslesen*)
VAR
	_sPkgName : STRING[10];
	_VerStruc : MoVerStruc_typ;
END_VAR
(*Aktueller Testmodus*)
VAR
	_wTestMode : UINT := 0;
END_VAR
(*Kommandointerpreter*)
VAR
	_CommandoState : _CommandoState_enum;
	_TestState : _TestState_enum;
	_fbSetMode : TestUser_SetMode;
	_fbRunTest : TestUser_RunTest;
	_doInfoCfg : DatObjInfo;
	_wMsgCnt : UINT;
	_MsgCfgList : REFERENCE TO ARRAY[1..MNMSG_MAX_CFGMESSAGES] OF MsgCfgLine_Typ;
	_ii : UINT;
END_VAR
VAR CONSTANT
	_MNTEST_MAX_MSGGROUPS : UINT := 30;
END_VAR
VAR
	_TONmsgclk2 : TON;
	_TONmsgclk1 : TON;
	_wMsgTick : UINT;
	_wStateMsgTest : ARRAY[1.._MNTEST_MAX_MSGGROUPS] OF UINT;
	_xReason : ARRAY[1.._MNTEST_MAX_MSGGROUPS] OF BOOL;
	_wMsgIdxOffset : ARRAY[1.._MNTEST_MAX_MSGGROUPS] OF UINT;
	_wMsgClass : ARRAY[0..4] OF UINT := [0,1,10,11,20];
	_TONMsg : ARRAY[1.._MNTEST_MAX_MSGGROUPS] OF TON;
	_TONMsgPause : ARRAY[1.._MNTEST_MAX_MSGGROUPS] OF TON;
END_VAR
```

#### _MessageTest1.st
```iecst
(********************************************************************
 * COPYRIGHT -- Herbert Kannegiesser GmbH
 ********************************************************************
 * Program: mnTest
 * File: _MessageTest1.st
 * Author: hunholz
 * Created: March 07, 2012
 ********************************************************************
 * Implementation of program mnTest
 ********************************************************************)

(* Meldungen zyklisch bearbeiten *)
ACTION _MessageTest1:

	_TONmsgclk1(IN := NOT _TONmsgclk2.Q, PT := T#15s);
	_TONmsgclk2(IN := _TONmsgclk1.Q, PT := T#15s);

	IF EDGEPOS(_TONmsgclk1.Q) THEN
		_wMsgTick := _wMsgTick + 1;
	END_IF

	IF _wMsgTick > _MNTEST_MAX_MSGGROUPS THEN
		_wMsgTick := 1;
	END_IF

	FOR _ii := 1 TO _MNTEST_MAX_MSGGROUPS DO

		CASE _wStateMsgTest[_ii] OF

			0:
				IF (_ii + _wMsgIdxOffset[_ii]) <= _wMsgCnt THEN
					// Warte auf Meldungsbeginn
					IF _ii = _wMsgTick THEN
						// Meldung setzen
						_xReason[_ii] := TRUE;
						kgMsgStatus[_ii].wFunction_ID := _MsgCfgList[_ii+_wMsgIdxOffset[_ii]].wFunction_ID;
						kgMsgStatus[_ii].wInstance := _MsgCfgList[_ii+_wMsgIdxOffset[_ii]].wInstance;

						IF _wMsgClass[_ii MOD 5] = MNMSG_CLASS_MAINTENANCE THEN
							kgMsgStatus[_ii].diMaintAttr1 := _ii;
							kgMsgStatus[_ii].diMaintAttr2 := _ii + 100;
							kgMsgStatus[_ii].sMaintAttrTxt := UINT_TO_STRING(_ii);
							kgMsgStatus[_ii].wMaintAckLevel := MNMSG_CLASS_NO_ACK;
							kgMsgStatus[_ii].wMaintNumber := _MsgCfgList[_ii+_wMsgIdxOffset[_ii]].wMsgNumber;
							kgMsgStatus[_ii].wMsgClass := MNMSG_CLASS_MAINTENANCE;
						ELSE
							kgMsgStatus[_ii].diMsgAttr1 := _ii;
							kgMsgStatus[_ii].diMsgAttr2 := _ii + 100;
							kgMsgStatus[_ii].sMsgAttrTxt := UINT_TO_STRING(_ii);
							kgMsgStatus[_ii].wMsgAckLevel := SEL((_wMsgClass[_ii MOD 4] < 10),0,MNMSG_CLASS_NO_ACK);
							kgMsgStatus[_ii].wMsgNumber := _MsgCfgList[_ii+_wMsgIdxOffset[_ii]].wMsgNumber;
							kgMsgStatus[_ii].wMsgClass := _wMsgClass[_ii MOD 5];
						END_IF

						_wStateMsgTest[_ii] := 1;

					END_IF
				ELSE
					_wMsgIdxOffset[_ii] := 0;
				END_IF

			1:
				// Warte bis Meldung beendet
				IF _TONMsg[_ii].Q THEN

					_xReason[_ii] := FALSE;

					IF kgMsgStatus[_ii].wMaintAckLevel = MNMSG_CLASS_NO_ACK THEN

						kgMsgStatus[_ii].wMaintAckLevel := _ii MOD 4;
						_wStateMsgTest[_ii] := 10;

					ELSIF kgMsgStatus[_ii].wMsgAckLevel = MNMSG_CLASS_NO_ACK THEN

						kgMsgStatus[_ii].wMsgAckLevel := _ii MOD 4;
						_wStateMsgTest[_ii] := 20;

					ELSE

						_wStateMsgTest[_ii] := 99;

					END_IF

				END_IF

			10:
			// Warten auf Wartungsquittierung

				IF kgMsgStatus[_ii].xAckMaint THEN
					kgMsgStatus[_ii].xAckRead := TRUE;
					_wStateMsgTest[_ii] := 99;
				END_IF

			20:
				// Warten auf Störungsquittierung

				IF kgMsgStatus[_ii].xAckFault THEN
					kgMsgStatus[_ii].xAckRead := TRUE;
					_wStateMsgTest[_ii] := 99;
				END_IF

			99:
				// Meldung entfernen
				kgMsgStatus[_ii].diMaintAttr1 := 0;
				kgMsgStatus[_ii].diMaintAttr2 := 0;
				kgMsgStatus[_ii].sMaintAttrTxt := '';
				kgMsgStatus[_ii].wMaintAckLevel := 0;
				kgMsgStatus[_ii].wMaintNumber := 0;
				kgMsgStatus[_ii].xAckRead := FALSE;
				kgMsgStatus[_ii].wMsgClass := 0;
				kgMsgStatus[_ii].diMsgAttr1 := 0;
				kgMsgStatus[_ii].diMsgAttr2 := 0;
				kgMsgStatus[_ii].sMsgAttrTxt := '';
				kgMsgStatus[_ii].wMsgAckLevel := 0;
				kgMsgStatus[_ii].wMsgNumber := 0;
				kgMsgStatus[_ii].wFunction_ID := 0;
				kgMsgStatus[_ii].wInstance := 0;

				_wStateMsgTest[_ii] := 100;

			100:
				// Warten bis Wartezeit beendet
				IF _TONMsgPause[_ii].Q THEN
					_wMsgIdxOffset[_ii] := _wMsgIdxOffset[_ii] + _MNTEST_MAX_MSGGROUPS;
					_wStateMsgTest[_ii] := 0;
				END_IF

		END_CASE

		_TONMsg[_ii](IN := _xReason[_ii], PT := T#10m);
		_TONMsgPause[_ii](IN := NOT _xReason[_ii], PT := T#4m);

	END_FOR

END_ACTION
```

### Package Logical/Mewa/KGFramework/Pkg_svCPCache - Category-Program-Verwaltung

### Pkg_svCPCache.typ - Global data types
```iecst
(********************************************************************
 * COPYRIGHT -- Herbert Kannegiesser GmbH
 ********************************************************************
 * Package: Pkg_svCPCache
 * File: Pkg_svCPCache.typ
 * Author: hunholz
 * Created: March 29, 2012
 ********************************************************************
 * Data types of package Pkg_svCPCache
 ********************************************************************)

TYPE
	svCPCache_Relation_Typ : 	STRUCT
		dtTimestamp : DATE_AND_TIME;
		sCategory : STRING[11];
		wProgramNo : UINT;
	END_STRUCT;
	IFsvCPCache_In_Typ : 	STRUCT
		wCmd : UINT;
		wReqUseDB : UINT;
		sReqCategory : STRING[11];
		utfReqCategoryName : WSTRING[31];
		wReqProgramNo : UINT;
		wReqLoadrate : UINT;
		rReqSoilfactor : REAL;
		wReqColidxFor : UINT;
		wReqColidxBack : UINT;
		wSetOffset : UINT;
	END_STRUCT;
	IFsvCPCache_Out_Typ : 	STRUCT
		xReady : BOOL;
		xListReady : BOOL;
		wCmdResponse : UINT;
		wCntRelations : UINT;
		wRespFromDB : UINT;
		utfRespCategoryName : WSTRING[31];
		rRespSoilFactor : REAL;
		wRespColidxFor : UINT;
		wRespColidxBack : UINT;
		wRespLoadrate : UINT;
		wRespProgramNo : UINT;
		utfRespProgramName : WSTRING[31];
		wListOffset : UINT;
		wListCnt : UINT;
		sListCategory : ARRAY[1..SVCPCACHE_CNT_LISTRELATIONS]OF STRING[11];
		utfListCategoryname : ARRAY[1..SVCPCACHE_CNT_LISTRELATIONS]OF WSTRING[31];
		wListProgramNo : ARRAY[1..SVCPCACHE_CNT_LISTRELATIONS]OF UINT;
		utfListProgramName : ARRAY[1..SVCPCACHE_CNT_LISTRELATIONS]OF WSTRING[31];
	END_STRUCT;
	IFsvCPCache_Typ : 	STRUCT
		In : IFsvCPCache_In_Typ;
		Out : IFsvCPCache_Out_Typ;
	END_STRUCT;
	svCPCacheStatAd_Typ : 	STRUCT
		xReady : BOOL;
		sPkgVersion : STRING[10];
	END_STRUCT;
END_TYPE
```

### Pkg_svCPCache.var - Global variables
```iecst
(********************************************************************
 * COPYRIGHT -- Herbert Kannegiesser GmbH
 ********************************************************************
 * Package: Pkg_svCPCache
 * File: Pkg_svCPCache.var
 * Author: hunholz
 * Created: March 29, 2012
 ********************************************************************
 * Variables of package Pkg_svCPCache
 ********************************************************************)
(*KONSTANTEN*)
VAR CONSTANT
	SVCPCACHE_DBREQ_LOCAL : UINT := 0;
	SVCPCACHE_DBREQ_DFII : UINT := 1;
END_VAR
(*Kommandos*)
VAR CONSTANT
	SVCPCACHE_CMD_GETPROG : UINT := 1;
	SVCPCACHE_CMD_INSERTCATEGORY : UINT := 2;
	SVCPCACHE_CMD_UPDATECATEGORY : UINT := 3;
	SVCPCACHE_CMD_DELETECATEGORY : UINT := 4;
	SVCPCACHE_CMD_SETOFFSET : UINT := 5;
END_VAR
(*Status*)
VAR CONSTANT
	SVCPCACHE_STAT_MEMALLOC : UINT := 60000;
	SVCPCACHE_STAT_CREATEFILE : UINT := 60001;
	SVCPCACHE_STAT_WRITEFILE : UINT := 60002;
	SVCPCACHE_STAT_OPENFILE : UINT := 60003;
	SVCPCACHE_STAT_NOSPACE : UINT := 60004;
	SVCPCACHE_STAT_INVALIDCATEGORY : UINT := 60005;
	SVCPCACHE_STAT_CATEGORYEXIST : UINT := 60006;
	SVCPCACHE_STAT_CATEGORYNOTEXIST : UINT := 60007;
	SVCPCACHE_STAT_CATEGORYLISTEMPTY : UINT := 60008;
	SVCPCACHE_STAT_DBNOTREADY : UINT := 60009;
END_VAR
(*Schnittstellen*)
VAR
	IFsvCPCache : IFsvCPCache_Typ;
	svCPCacheStatAd : svCPCacheStatAd_Typ;
END_VAR
```

### Program Logical/Mewa/KGFramework/Pkg_svCPCache/svCPCache (IEC) - Category-Program-Cache

#### svCPCacheCyclic.st - Cyclic code
```iecst
(********************************************************************
 * COPYRIGHT -- Herbert Kannegiesser GmbH
 ********************************************************************
 * Program: svCPCache
 * File: svCPCacheCyclic.st
 * Author: hunholz
 * Created: March 29, 2012
 ********************************************************************
 * Implementation of program svCPCache
 ********************************************************************)

PROGRAM _CYCLIC

	// Zyklische Arbeit. Entgegennehmen von Aufträgen
	IF _xCacheReady THEN

		// Kommandos abarbeiten
		_actIFCmd;

		// CSV-File speichern
		_actSaveCSV;

	END_IF

	// Erstmaliges Lesen der Kategorie-Programm-Zuordnung
	IF _xCacheInitReady AND NOT _xCacheReady AND IFmnParam.Out.xParamOK THEN

		IF _enImport = cs_ImpIdle THEN
			_enImport := cs_ImpStart;
		END_IF

		///////////////////////////////
		// ACTION
		///////////////////////////////
		_actCPImport;

		IF _enImport = cs_ImpRdyFault THEN

			// Einlesen mit Fehler abgebrochen
			_xCacheInitReady := FALSE;

			_enImport := cs_ImpIdle;

		ELSIF _enImport = cs_ImpRdySuccess THEN

			// Erfolgreich eingelesen
			_xCacheReady := TRUE;

			IFsvCPCache.Out.xListReady := TRUE;
			IFsvCPCache.Out.wCntRelations := _wCntRelations;

			// Liste füllen
			IFsvCPCache.Out.wListOffset := 0;
			_actFillCPList;

			_enImport := cs_ImpIdle;

		END_IF

	END_IF

	IFsvCPCache.Out.xReady := _xCacheReady;
	svCPCacheStatAd.xReady := _xCacheReady;

END_PROGRAM
```

#### svCPCacheInit.st - Initialization code
```iecst
(********************************************************************
 * COPYRIGHT -- Herbert Kannegiesser GmbH
 ********************************************************************
 * Program: svCPCache
 * File: svCPCacheInit.st
 * Author: hunholz
 * Created: March 29, 2012
 ********************************************************************
 * Implementation of program svCPCache
 ********************************************************************)

PROGRAM _INIT

	// Packet-Version auslesen mit MO_ver aus SYS_lib und für den Additional Status zur Verfügung stellen

	_sPkgName := 'svCPCache';

	IF ( MO_ver(ADR(_sPkgName), 0, ADR(_VerStruc)) = 0 ) THEN

		brsmemcpy(ADR(svCPCacheStatAd.sPkgVersion), ADR(_VerStruc.version), SIZEOF(_VerStruc.version));

	ELSE

		svCPCacheStatAd.sPkgVersion := '---';

	END_IF

	_xCacheInitReady := FALSE;

	REPEAT // UNTIL TRUE

		// Schleife, die nur einmal durchlaufen wird, aber jederzeit verlassen werden kann

		//Mögliche Optionen
		//SVCPCACHE_DBREQ_NO = 0
		//SVCPCACHE_DBREQ_DFII = 1
		IF SVCPCACHE_DB_REQUEST > 1 THEN
			EXIT;
		END_IF

		//Container sind von 0..20 möglich
		IF SVCPCACHE_NO_INDCONTAINER > 20 THEN
			EXIT;
		END_IF

		// Speicher zum Parsen und Schreiben allokieren

		_lMemLen := SVCPCACHE_CNT_RELATIONS * 146 + 200;

		_MemPartCreate(enable := TRUE, len := _lMemLen + 100);

		IF _MemPartCreate.status <> ERR_OK THEN
			EXIT;
		END_IF

		_xCacheInitReady := TRUE;

		UNTIL TRUE

	END_REPEAT

END_PROGRAM
```

#### svCPCache.typ - Local data types
```iecst
(********************************************************************
 * COPYRIGHT -- Herbert Kannegiesser GmbH
 ********************************************************************
 * Program: svCPCache
 * File: svCPCache.typ
 * Author: hunholz
 * Created: March 29, 2012
 ********************************************************************
 * Local data types of program svCPCache
 ********************************************************************)

TYPE
	enum_CmdCP :
		(
		cs_CmdIdle,
		cs_CmdSave,
		cs_CmdWaitForDB,
		cs_CmdWaitForNoCommand
		);
	enum_ImportCP :
		(
		cs_ImpIdle,
		cs_ImpStart,
		cs_ImpFileOpen,
		cs_ImpFileRead,
		cs_ImpFileClose,
		cs_ImpParse,
		cs_ImpRdySuccess,
		cs_ImpRdyFault
		);
	enum_SaveCP :
		(
		cs_SaveIdle,
		cs_SaveCreateCSV,
		cs_SaveDeleteFile,
		cs_SaveCreateFile,
		cs_SaveOpenFile,
		cs_SaveWriteFile,
		cs_SaveCloseFile,
		cs_SaveRdySuccess,
		cs_SaveRdyFault
		);
END_TYPE
```

#### svCPCache.var - Local variables
```iecst
(********************************************************************
 * COPYRIGHT -- Herbert Kannegiesser GmbH
 ********************************************************************
 * Program: svCPCache
 * File: svCPCache.var
 * Author: hunholz
 * Created: March 29, 2012
 ********************************************************************
 * Local variables of program svCPCache
 ********************************************************************)
VAR CONSTANT
	_SVCPCACHE_CSV_FILE : STRING[31] := 'PM\Export\cpcache.csv';
END_VAR
VAR
	_sPkgName : STRING[11];
	_VerStruc : MoVerStruc_typ;
	_CPCache : ARRAY[1..SVCPCACHE_CNT_RELATIONS] OF mnParam_CProw_typ;
	_wCntRelations : UINT;
	_i : UINT;
	_lMemLen : UDINT;
	_lLineAdress : ARRAY[1..SVCPCACHE_MAX_PARSELINES] OF UDINT;
	_wLineLen : ARRAY[1..SVCPCACHE_MAX_PARSELINES] OF UINT;
	_wStartLine : UINT;
	_CountLines : mnParam_CountLines;
	_GetCsvDat : mnParam_GetCsvDat;
	_enCmd : enum_CmdCP;
	_enImport : enum_ImportCP;
	_enSave : enum_SaveCP;
	_xImpFault : BOOL;
	_xImpReady : BOOL;
	_MemPartCreate : AsMemPartCreate;
	_FileOpen : FileOpen;
	_FileRead : FileRead;
	_FileClose : FileClose;
	_MemPartAllocClear : AsMemPartAllocClear;
	_MemPartFree : AsMemPartFree;
	_lTempMem : UDINT;
	_lFileLen : UDINT;
	_xCacheInitReady : BOOL;
	_xCacheReady : BOOL;
	_wfcli : UINT;
	_wfclj : UINT;
	_SaveMemPartAlloc : AsMemPartAllocClear;
	_lWriteSize : UDINT;
	_WriteBOM : mnParam_WriteBOM_Mem;
	_WriteComment : mnParam_WriteCSV254_Mem;
	_WriteNewLine : mnParam_WriteNewline_Mem;
	_MachineNoRow : mnParam_HeaderMachineNoRow_typ;
	_WriteMachineNo : mnParam_WriteCSV252_Mem;
	_DTGetTime : DTGetTime;
	_HeaderTimeRow : mnParam_HeaderTimeRow_typ;
	_WriteTimeStamp : mnParam_WriteCSV251_Mem;
	_sci : UINT;
	_WriteCP : mnParam_WriteCSV81_Mem;
	_FileCreate : FileCreate;
	_FileDelete : FileDelete;
	_wSaveCSVstatus : UINT;
	_SaveMemPartFree : AsMemPartFree;
	_FileWrite : FileWrite;
	_sCategory : STRING[11];
	_xCategoryExist : BOOL;
	_wCmd : UINT;
	_TrimCat : _TrimCategory;
	_wCategoryIdx : UINT;
END_VAR
```

#### _actCPImport.st
```iecst
(********************************************************************
 * COPYRIGHT -- Herbert Kannegiesser GmbH
 ********************************************************************
 * Program: svCPCache
 * File: _actCPImport.st
 * Author: hunholz
 * Created: March 29, 2012
 ********************************************************************
 * Implementation of program svCPCache
 ********************************************************************)

(* Kategorie-Programm-Zuordnung aus CSV-Datei lesen *)
ACTION _actCPImport:

	CASE _enImport OF

		cs_ImpIdle:

			// Tue nichts

		cs_ImpStart:

			// Initialisierung
			brsmemset(ADR(_CPCache), 0, SIZEOF(_CPCache));
			brsmemset(ADR(_lLineAdress), 0, SIZEOF(_lLineAdress));
			brsmemset(ADR(_wLineLen), 0, SIZEOF(_wLineLen));
			_wCntRelations := 0;
			_xImpFault := FALSE;
			_xImpReady := FALSE;
			_lTempMem := 0;

			_enImport := cs_ImpFileOpen;

		cs_ImpFileOpen:

			_FileOpen(enable := TRUE, pDevice := ADR(KG_DEVICE_COMPACTFLASH), pFile := ADR(_SVCPCACHE_CSV_FILE), mode := fiREAD_ONLY);

			IF _FileOpen.status = ERR_OK THEN

				IF _FileOpen.filelen > SIZEOF(KGBOM) THEN

					_lFileLen := _FileOpen.filelen - SIZEOF(KGBOM);

					_MemPartAllocClear(enable := TRUE, ident := _MemPartCreate.ident, len := _lFileLen);

					IF _MemPartAllocClear.status = ERR_OK THEN

						_lTempMem := _MemPartAllocClear.mem;
						_enImport := cs_ImpFileRead;

					ELSE

						_xImpFault := TRUE;
						_enImport := cs_ImpFileClose;

					END_IF

				ELSE

					_xImpReady := TRUE;
					_enImport := cs_ImpFileClose;

				END_IF

			ELSIF _FileOpen.status <> ERR_FUB_BUSY THEN

				_enImport := cs_ImpRdySuccess;

			END_IF

		cs_ImpFileRead:

			_FileRead(enable := TRUE, ident := _FileOpen.ident, offset := SIZEOF(KGBOM), pDest := _MemPartAllocClear.mem, len := _lFileLen);

			IF _FileRead.status <> ERR_FUB_BUSY THEN

				IF _FileRead.status <> ERR_OK THEN

					_xImpFault := TRUE;

				END_IF

				_enImport := cs_ImpFileClose;

			END_IF

		cs_ImpFileClose:

			_FileClose(enable := TRUE, ident := _FileOpen.ident);

			IF _FileClose.status = ERR_OK THEN

				IF _xImpFault THEN

					_enImport := cs_ImpRdyFault;

					IF _lTempMem <> 0 THEN
						_MemPartFree(enable := TRUE, ident := _MemPartAllocClear.ident, mem := _lTempMem);
					END_IF

				ELSIF _xImpReady THEN

					_enImport := cs_ImpRdySuccess;

					IF _lTempMem <> 0 THEN
						_MemPartFree(enable := TRUE, ident := _MemPartAllocClear.ident, mem := _lTempMem);
					END_IF

				ELSE

					_enImport := cs_ImpParse;

				END_IF

			ELSIF _FileClose.status <> ERR_FUB_BUSY THEN

				_enImport := cs_ImpRdyFault;

			END_IF

		cs_ImpParse:

			_CountLines.enable 	:= TRUE;
			_CountLines.pFile 		:= _lTempMem;
			_CountLines.FileSize 	:= _lFileLen;
			_CountLines.MaxLines	:= SVCPCACHE_MAX_PARSELINES;
			_CountLines.pAdresses	:= ADR(_lLineAdress);
			_CountLines.pLens		:= ADR(_wLineLen);

			_CountLines();

			IF _CountLines.status <> ERR_OK THEN

				_MemPartFree(enable := TRUE, ident := _MemPartAllocClear.ident, mem := _lTempMem);
				_enImport := cs_ImpRdyFault;

			ELSE

				_wStartLine := 1;

				REPEAT

					_GetCsvDat.enable := TRUE;
					brwcsncpy( ADR(_GetCsvDat.utfCsvString), _lLineAdress[_wStartLine], MIN(299, _wLineLen[_wStartLine]));
					_GetCsvDat();

					IF _GetCsvDat.RowType = MNPARAM_CSV_CP AND _wCntRelations < SVCPCACHE_CNT_RELATIONS THEN

						_wCntRelations := _wCntRelations + 1;

						_CPCache[_wCntRelations] := _GetCsvDat.CsvCProw;

					END_IF

					_wStartLine := _wStartLine + 1;

					UNTIL
					_wStartLine > _CountLines.CntLines

				END_REPEAT

				_MemPartFree(enable := TRUE, ident := _MemPartAllocClear.ident, mem := _lTempMem);
				_enImport := cs_ImpRdySuccess;

			END_IF

		cs_ImpRdySuccess:

			// Beendet mit Erfolg

		cs_ImpRdyFault:

			// Mit Fehler beendet

	END_CASE

END_ACTION
```
